# B&R Automation Studio project Parker_BMM_ST_V5_3147_V12 (part 12)

#### bdeflash.c
```c
/********************************************************************
 * COPYRIGHT --  B&R China
 ********************************************************************
 * Program: bdeflash
 * File: bdeflash.c
 * Author: lijianjun
 * Created: March 06, 2013
 ********************************************************************
 * Implementation of program bdeflash --- bottom deflasher control
 ********************************************************************/

#include <bur/plctypes.h>

#ifdef _DEFAULT_INCLUDES
	#include <AsDefault.h>
#endif

/**************************************************************************************
                            Function Declarations
**************************************************************************************/

//void BottomDeflash( Mold_typ * pMold);
void BottomDeflash( Mold_typ * pMold,TopDeflash_Fix_typ * pBottomDeflashFix, TopDeflash_Para_typ * pBottomDeflashPara,Mold_Para_User_typ * pMoldUser);
/**************************************************************************************
     	        		I N I T U P  O F   T H E   T A S K
**************************************************************************************/
_INIT void init ( void )
 {
 	LMold.BottomDeflash.Step = 0;
 	RMold.BottomDeflash.Step = 0;
 } /* end of _INIT */

 /*************************************************************************************
        		底部去飞边		C Y C L I C   P A R T   O F   T H E   T A S K
**************************************************************************************/

 _CYCLIC void cyclic ( void )
 {
 	if(!LMold.TimeSet.BottomDeflashBwAlarmTime)LMold.TimeSet.BottomDeflashBwAlarmTime = 1000;  /*  10s  */
 	if(!RMold.TimeSet.BottomDeflashBwAlarmTime)RMold.TimeSet.BottomDeflashBwAlarmTime = 1000;  /*  10s  */

 	LMold.TransDIn.BottomDeflashBwLimit = gMachineIn.LMold.BottomDeflashBwLimit;
 	LMold.TransDIn.BottomDeflashFwLimit = gMachineIn.LMold.BottomDeflashFwLimit;

	RMold.TransDIn.BottomDeflashBwLimit = gMachineIn.RMold.BottomDeflashBwLimit;
	RMold.TransDIn.BottomDeflashFwLimit = gMachineIn.RMold.BottomDeflashFwLimit;

	BottomDeflash(&LMold,&gMachineFix.MoldL.BottomDeflash,&gMachinePara.MoldL.BottomDeflash,&gUserPara.LMold);
	BottomDeflash(&RMold,&gMachineFix.MoldR.BottomDeflash,&gMachinePara.MoldR.BottomDeflash,&gUserPara.RMold);

//	gMachineOut.LMold.BottomDeflashFw = LMold.BottomDeflash.Out;
//	gMachineOut.RMold.BottomDeflashFw = RMold.BottomDeflash.Out;

	gMachineOut.LMold.BottomDeflashFw = LMold.ValveOut.BottomDeflashFw;
	gMachineOut.RMold.BottomDeflashFw = RMold.ValveOut.BottomDeflashFw;

	gMachineOut.LMold.BottomDeflashBw = LMold.ValveOut.BottomDeflashBw;
	gMachineOut.RMold.BottomDeflashBw = RMold.ValveOut.BottomDeflashBw;

	/*------------- ActuatorType--------------- */
	gMachineFix.MoldL.BottomDeflash.eActuatorType = gMachineFix.MoldR.BottomDeflash.eActuatorType;

	/*------------ PressueOutputType--------------- */
	gMachineFix.MoldL.BottomDeflash.ePressueOutputType = gMachineFix.MoldR.BottomDeflash.ePressueOutputType;

	/*------------ FluxOutputType--------------- */
	gMachineFix.MoldL.BottomDeflash.eFluxOutputType = gMachineFix.MoldR.BottomDeflash.eFluxOutputType;

 } /* end of _CYCLIC */

void BottomDeflash( Mold_typ * pMold,TopDeflash_Fix_typ * pBottomDeflashFix, TopDeflash_Para_typ * pBottomDeflashPara,Mold_Para_User_typ * pMoldUser)
{

	switch ( pMold->BottomDeflash.Step )
	{
		/*------------------ stop all the output ------------------*/
		case 0:
			pMold->BottomDeflash.Out      = 0;
			pMold->ActInfo.BottomDeflash  = 0;
			pMold->ActInfo.BottomDeflashFw  = 0;
			pMold->ActInfo.BottomDeflashBw  = 0;

			pMold->ValveOut.BottomDeflashFw = 0;

			if (0 == gMachineInfo.Auto)
			{
				pMold->ValveOut.BottomDeflashBw = 0;//ipis0726
			}

			pMold->BottomDeflash.Timer.IN	= 0;
			break;

		/*------------------ TopDeflash forward -------------------- */
		case 90: 			/* forward  Extra delay for Extrilift Acc charge */
			if(pMold->Option.BottomDeflash)
			{
				if(pMoldUser->TimeSet.BottomDeflashExtraDelay != 0)
				{
					pMold->BottomDeflash.Timer.IN = 1;
					pMold->BottomDeflash.Timer.PT = pMoldUser->TimeSet.BottomDeflashExtraDelay;
					pMold->BottomDeflash.Step 	= 95;
				}
				else
				{
					pMold->BottomDeflash.Step = 100;
				}
			}
			else
			{
				pMold->BottomDeflash.Step = 100;
			}

			break;

		case 95: 	/*Extara delay*/
			pMoldUser->TimeDis.BottomDeflashExtraDelay = pMold->BottomDeflash.Timer.ET;
			if (1 == pMold->BottomDeflash.Timer.Q)
			{
				pMold->BottomDeflash.Timer.IN       = 0;
				//	pMold->TimeDis.TopDeflashFwDelay = 0;
				pMold->BottomDeflash.Step = 100;
			}

			break;

		/*------------------ BottomDeflash forward -------------------- */
		case 100: /* BottomDeflash delay*/

			if(pMold->Option.BottomDeflash)
			{
				if(pMold->TimeSet.BottomDeflashFwDelay != 0)
				{
					pMold->BottomDeflash.Timer.IN = 1;
					pMold->BottomDeflash.Timer.PT = pMold->TimeSet.BottomDeflashFwDelay;
					pMold->BottomDeflash.Step 	= 200;
				}
				else
				{
					pMold->BottomDeflash.Step = 300;
				}
			}
			else
			{
				pMold->BottomDeflash.Step = 300;
			}
			break;

		case 200: 		/* delay ok */
			pMold->TimeDis.BottomDeflashFwDelay = pMold->BottomDeflash.Timer.ET;
			if (1 == pMold->BottomDeflash.Timer.Q)
			{
				pMold->BottomDeflash.Timer.IN       = 0;
				//	pMold->TimeDis.BottomDeflashFwDelay = 0;
				pMold->BottomDeflash.Step = 300;
			}
			break;

		case 300:
			if(pMold->Option.BottomDeflash)
			{
				switch (pBottomDeflashFix->eActuatorType )
				{
					/*-------------------------------------------------*/
					case ACTUATOR_HYD: /*1:Oil*/
					/*-------------------------------------------------*/
						if(pMold->TimeSet.BottomDeflashFwTime != 0 )
						{
							pMold->BottomDeflash.LimitTimer.IN = 1; //ipis0213
							pMold->BottomDeflash.LimitTimer.PT = pMold->TimeSet.BottomDeflashFwAlarmTime;

							pMold->BottomDeflash.Timer.IN = 1;
							pMold->BottomDeflash.Timer.PT = pMold->TimeSet.BottomDeflashFwTime;
							pMold->BottomDeflash.Step = 400;
						}
						else
						{
							//	pMold->BottomDeflash.Step = 499;
							pMold->BottomDeflash.Step = 2900; //ipis 0213
						}
						break;
					/*-------------------------------------------------*/
					case ACTUATOR_PNEU: /*2:Air*/
					/*-------------------------------------------------*/
						if(pMold->TimeSet.BottomDeflashFwTime != 0 )
						{
							pMold->BottomDeflash.Timer.IN = 1;
							pMold->BottomDeflash.Timer.PT = pMold->TimeSet.BottomDeflashFwTime;
							pMold->BottomDeflash.Step = 400;
						}
						else
						{
							//	pMold->BottomDeflash.Step = 499;
							pMold->BottomDeflash.Step = 2900; //ipis 0213
						}
						break;
				}
			}
			else
			{
				pMold->BottomDeflash.Step = 2900; // for no use
			}

			break;

		case 400:			/* forward time ok */
			pMold->BottomDeflash.Out     = 1;
			pMold->ActInfo.BottomDeflash = 1;
			pMold->ActInfo.BottomDeflashFw  = 1;
			pMold->ActInfo.BottomDeflashBw  = 0;

			pMold->ValveOut.BottomDeflashFw = 1;
			pMold->ValveOut.BottomDeflashBw = 0;

			pMold->BottomDeflash.p_set = pBottomDeflashPara->P_Fw;

			pMold->TimeDis.BottomDeflashFwTime = pMold->BottomDeflash.Timer.ET;

			if ((1 == pMold->BottomDeflash.Timer.Q) )
			{

				pMold->BottomDeflash.Out      = 0;
				pMold->ActInfo.BottomDeflashFw  = 0;
				pMold->ActInfo.BottomDeflashBw  = 0;

				pMold->ValveOut.BottomDeflashFw = 0;
				pMold->ValveOut.BottomDeflashBw = 0;

				pMold->BottomDeflash.p_set = 0;
				pMold->BottomDeflash.Timer.IN = 0;
				pMold->BottomDeflash.LimitTimer.IN = 0;
				//	pMold->TimeDis.BottomDeflashFwTime = 0;

				pMold->BottomDeflash.Step     = 410;

			}

			pMold->TimeDis.BottomDeflashFwAlarmTime = pMold->BottomDeflash.LimitTimer.ET;

			break;

		/*------------------------------------------------------------------------------*/

		case 410:/*Second Forward Delay*/

			switch (pBottomDeflashFix->eActuatorType)
			{
				/*-------------------------------------------------*/
				case ACTUATOR_HYD: /*1:Oil*/
				/*-------------------------------------------------*/
					if(pMoldUser->TimeSet.BottomDeflashSecDelay != 0)
					{
						pMold->BottomDeflash.Timer.IN = 1;
						pMold->BottomDeflash.Timer.PT = pMoldUser->TimeSet.BottomDeflashSecDelay;
						pMold->BottomDeflash.Step = 420;
					}
					else
					{
						pMold->BottomDeflash.Step = 430;
					}
					break;
				/*-------------------------------------------------*/
				case ACTUATOR_PNEU: /*2:Air*/
				/*-------------------------------------------------*/
					pMold->BottomDeflash.Step = 1300;
					break;
			}
			break;
		case 420: /*Start Second TopDeflash Forward Timer*/

			pMold->BottomDeflash.Out      = 0;
			pMold->ActInfo.BottomDeflashFw  = 0;
			pMold->ActInfo.BottomDeflashBw  = 0;

			pMold->ValveOut.BottomDeflashFw = 0;
			pMold->ValveOut.BottomDeflashBw = 0;

			pMold->BottomDeflash.p_set = 0;

			pMoldUser->TimeDis.BottomDeflashSecDelay = pMold->BottomDeflash.Timer.ET;
			if (1 == pMold->BottomDeflash.Timer.Q)
			{
				pMold->BottomDeflash.Timer.IN       = 0;
				pMold->BottomDeflash.LimitTimer.IN 	= 0;
				//	pMoldUser->TimeDis.BottomDeflashSecDelay = 0;
				pMold->BottomDeflash.Step = 430;
			}
			break;

		case 430:		/*Start Second TopDeflash Forward Timer*/
			if(pMoldUser->TimeSet.BottomDeflashSecTime != 0)
			{
				pMold->BottomDeflash.LimitTimer.IN = 1; //ipis0213
				pMold->BottomDeflash.LimitTimer.PT = pMold->TimeSet.BottomDeflashFwAlarmTime;

				pMold->BottomDeflash.Timer.IN = 1;
				pMold->BottomDeflash.Timer.PT = pMoldUser->TimeSet.BottomDeflashSecTime;
				pMold->BottomDeflash.Step = 440;
			}
			else
			{
				pMold->BottomDeflash.Step = 1300;
			}
			break;

		case 440:  /*Bottom deflash second forward */
			pMold->BottomDeflash.Out     = 1;
			pMold->ActInfo.BottomDeflash = 1;
			pMold->ActInfo.BottomDeflashFw  = 1;
			pMold->ActInfo.BottomDeflashBw  = 0;

			pMold->ValveOut.BottomDeflashFw = 1;
			pMold->ValveOut.BottomDeflashBw = 0;

			pMold->BottomDeflash.p_set = pBottomDeflashPara->P_Fw2nd;

			pMoldUser->TimeDis.BottomDeflashSecTime = pMold->BottomDeflash.Timer.ET;
			if ((1 == pMold->BottomDeflash.Timer.Q) || (1 == pMold->TransDIn.BottomDeflashFwLimit))
			{

				pMold->BottomDeflash.Out      = 0;
				pMold->ActInfo.BottomDeflashFw  = 0;
				pMold->ActInfo.BottomDeflashBw  = 0;

				pMold->ValveOut.BottomDeflashFw = 0;
				pMold->ValveOut.BottomDeflashBw = 0;
				pMold->BottomDeflash.p_set = 0;
				pMold->BottomDeflash.Timer.IN = 0;
				//	pMold->TimeDis.BottomDeflashFwTime = 0;
				//	pMoldUser->TimeDis.BottomDeflashSecTime=0;
				pMold->BottomDeflash.Step     = 1300;
			}
			pMold->TimeDis.BottomDeflashFwAlarmTime = pMold->BottomDeflash.LimitTimer.ET;

			break;

		/*----------------------------------------------*/
		/*No Time Movement-move unitl reach limit sensor*/
		/*----------------------------------------------*/

		case 499:
			pMold->BottomDeflash.Out     = 1;
			pMold->ActInfo.BottomDeflash = 1;
			pMold->ActInfo.BottomDeflashFw  = 1;
			pMold->ActInfo.BottomDeflashBw  = 0;

			pMold->ValveOut.BottomDeflashFw = 1;
			pMold->ValveOut.BottomDeflashBw = 0;

			pMold->BottomDeflash.p_set = pBottomDeflashPara->P_Fw;

			if (1 == pMold->TransDIn.BottomDeflashFwLimit)
			{

				pMold->BottomDeflash.Out      = 0;
				pMold->ActInfo.BottomDeflashFw  = 0;
				pMold->ActInfo.BottomDeflashBw  = 0;

				pMold->ValveOut.BottomDeflashFw = 0;
				pMold->ValveOut.BottomDeflashBw = 0;
				pMold->BottomDeflash.p_set = 0;
				pMold->BottomDeflash.Timer.IN = 0;
				pMold->BottomDeflash.LimitTimer.IN = 0;
				//	pMold->TimeDis.BottomDeflashFwTime = 0;

				pMold->BottomDeflash.Step     = 2900;
			}

			pMold->TimeDis.BottomDeflashFwAlarmTime = pMold->BottomDeflash.LimitTimer.ET;

			if (1 == pMold->BottomDeflash.LimitTimer.Q )
			{
				pMold->Alarm.BottomDeflashNotAtFwPos=1;
				pMold->BottomDeflash.Timer.IN   = 0;
				pMold->BottomDeflash.LimitTimer.IN = 0;
				pMold->BottomDeflash.Step = 40000;
			}

			break;

		case 1000:
			pMold->BottomDeflash.Out     = 1;
			pMold->ActInfo.BottomDeflashFw  = 1;
			pMold->ActInfo.BottomDeflashBw  = 0;
			pMold->BottomDeflash.p_set = pBottomDeflashPara->P_Fw;
			pMold->ValveOut.BottomDeflashFw = 1;
			pMold->ValveOut.BottomDeflashBw = 0;

			pMold->ActInfo.BottomDeflash = 1;
			break;

		/*------- BottomDeflash Bw --------------------------*/

		case 1300: /* BottomDeflash Bw delay*/
			if(pMold->Option.BottomDeflash)
			{
				switch (pBottomDeflashFix->eActuatorType)
				{
					/*-------------------------------------------------*/
					case ACTUATOR_HYD: /*1:Oil*/
					/*-------------------------------------------------*/
						if(pMold->TimeSet.BottomDeflashBwDelay != 0)
						{
							pMold->BottomDeflash.Timer.IN = 1;
							pMold->BottomDeflash.Timer.PT = pMold->TimeSet.BottomDeflashBwDelay;
							pMold->BottomDeflash.Step 	= 1400;
						}
						else
						{
							pMold->BottomDeflash.Step = 1500;
						}

						break;
					/*-------------------------------------------------*/
					case ACTUATOR_PNEU: /*2:Air*/
					/*-------------------------------------------------*/
						pMold->BottomDeflash.Step = 1500;
						break;
				}
			}
			else
			{
				pMold->BottomDeflash.Step = 1500;
			}
			break;
		case 1400: /* delay ok */
			pMold->TimeDis.BottomDeflashBwDelay = pMold->BottomDeflash.Timer.ET;
			if (1 == pMold->BottomDeflash.Timer.Q)
			{
				pMold->BottomDeflash.Timer.IN       = 0;
				//		pMold->TimeDis.BottomDeflashBwDelay = 0;
				pMold->BottomDeflash.Step = 1500;
			}
			break;

		case 1500:

			if(pMold->Option.BottomDeflash)
			{
				pMold->BottomDeflash.Timer.IN = 1;
				pMold->BottomDeflash.Timer.PT = pMold->TimeSet.BottomDeflashBwAlarmTime;
				pMold->BottomDeflash.Step = 1600;
			}
			else
			{
				pMold->BottomDeflash.Step = 1700; // for no use
			}
			break;

		case 1600:
			pMold->BottomDeflash.Out     = 0;

			pMold->ActInfo.BottomDeflash = 0;
			pMold->ActInfo.BottomDeflashFw  = 0;
			pMold->ActInfo.BottomDeflashBw  = 1;

			pMold->ValveOut.BottomDeflashFw = 0;
			pMold->ValveOut.BottomDeflashBw = 1;

			pMold->BottomDeflash.p_set = pBottomDeflashPara->P_Bw;

			pMold->TimeDis.BottomDeflashBwAlarmTime = pMold->BottomDeflash.Timer.ET;

			if (1 == pMold->TransDIn.BottomDeflashBwLimit)
			{
				pMold->BottomDeflash.Out      = 0;
				pMold->ActInfo.BottomDeflashFw  = 0;
				pMold->ActInfo.BottomDeflashBw  = 0;

				pMold->ValveOut.BottomDeflashFw = 0;
				pMold->ValveOut.BottomDeflashBw = 0;
				pMold->BottomDeflash.p_set=0;

				pMold->BottomDeflash.Timer.IN = 0;
				pMold->TimeDis.BottomDeflashBwTime = 0;
				pMold->BottomDeflash.Step     = 2900;
			}

			break;

		case 1700: // for no use

			if (1 == pMold->TransDIn.BottomDeflashBwLimit)
			{
				pMold->BottomDeflash.Out      = 0;
				pMold->ActInfo.BottomDeflashFw  = 0;
				pMold->ActInfo.BottomDeflashBw  = 0;

				pMold->ValveOut.BottomDeflashFw = 0;
				pMold->ValveOut.BottomDeflashBw = 0;
				pMold->BottomDeflash.p_set=0;

				pMold->BottomDeflash.Timer.IN = 0;
				pMold->TimeDis.BottomDeflashBwTime = 0;
				pMold->BottomDeflash.Step     = 2900;
			}
			else
			{
				pMold->BottomDeflash.Timer.IN   = 0;
				pMold->Alarm.BottomDeflashNotAtBwPos = 1;
				pMold->BottomDeflash.Step = 40000;           /*  TopDeflash backward alarm   */

			}

			//			pMold->TimeDis.BottomDeflashBwAlarmTime = pMold->BottomDeflash.Timer.ET;
			//			if(1 == pMold->BottomDeflash.Timer.Q)
			//			{
			//				pMold->ValveOut.BottomDeflashFw  = 0;
			//				pMold->ValveOut.BottomDeflashBw  = 0;
			//
			//				pMold->BottomDeflash.Timer.IN   = 0;
			//				pMold->Alarm.BottomDeflashNotAtBwPos = 1;
			//				pMold->BottomDeflash.Step = 40000;           /*  TopDeflash backward alarm   */
			//			}

			break;
		/*----------for handle bottom deflash force backward------------------------------*/
		case 1950: //for auto force backward

			pMold->BottomDeflash.Timer.IN = 0;
			pMold->BottomDeflash.LimitTimer.IN = 0;
			pMold->BottomDeflash.Step = 2000;

			break;

		case 2000:
			pMold->BottomDeflash.Out     = 0;
			pMold->ActInfo.BottomDeflash = 0;
			pMold->ActInfo.BottomDeflashFw  = 0;
			pMold->ActInfo.BottomDeflashBw  = 0;
			pMold->BottomDeflash.p_set=0;
			pMold->ValveOut.BottomDeflashFw = 0;
			pMold->ValveOut.BottomDeflashBw = 0;

			pMold->BottomDeflash.Step    = 0;
			break;

		case 2900:

			pMold->BottomDeflash.Timer.IN = 0;
			pMold->BottomDeflash.LimitTimer.IN = 0;
			pMold->BottomDeflash.Out     = 0;
			pMold->ActInfo.BottomDeflashFw  = 0;
			pMold->ActInfo.BottomDeflashBw  = 0;
			pMold->BottomDeflash.p_set=0;

			pMold->ValveOut.BottomDeflashFw = 0;
			pMold->ValveOut.BottomDeflashBw = 0;
			pMold->ActInfo.BottomDeflash = 0;
			pMold->BottomDeflash.Step    = 3000;
			break;

		case 3000:
			break;

		case 5000: /* FW*/

			//			pMold->ActInfo.BottomDeflashFw  = 1;
			//			pMold->ActInfo.BottomDeflashBw  = 0;
			//
			//			pMold->ValveOut.BottomDeflashFw = 1;
			//			pMold->ValveOut.BottomDeflashBw = 0;
			//
			//			pMold->BottomDeflash.p_set = pBottomDeflashPara->P_CalibFw;

			if(0 == pMold->TransDIn.BottomDeflashFwLimit)
			{
				pMold->ActInfo.BottomDeflashFw  = 1;
				pMold->ActInfo.BottomDeflashBw  = 0;

				pMold->ValveOut.BottomDeflashFw = 1;
				pMold->ValveOut.BottomDeflashBw = 0;

				pMold->BottomDeflash.p_set = pBottomDeflashFix->pCalibMax;
				pMold->BottomDeflash.v_set = pBottomDeflashFix->vCalibMax;
			}
			else
			{
				pMold->ActInfo.BottomDeflashFw  = 0;
				pMold->ActInfo.BottomDeflashBw  = 0;

				pMold->ValveOut.BottomDeflashFw = 0;
				pMold->ValveOut.BottomDeflashBw = 0;

				pMold->BottomDeflash.p_set 		= 0;
				pMold->BottomDeflash.v_set		= 0;

				pMold->BottomDeflash.Step    	= 20000;
			}

			break;

		case 15000: /* BW*/

			//			pMold->ActInfo.BottomDeflashFw  = 0;
			//			pMold->ActInfo.BottomDeflashBw  = 1;
			//
			//			pMold->ValveOut.BottomDeflashFw = 0;
			//			pMold->ValveOut.BottomDeflashBw = 1;
			//
			//			pMold->BottomDeflash.p_set = pBottomDeflashPara->P_CalibBw;

			if(0 == pMold->TransDIn.BottomDeflashBwLimit)
			{
				pMold->ActInfo.BottomDeflashFw  = 0;
				pMold->ActInfo.BottomDeflashBw  = 1;

				pMold->ValveOut.BottomDeflashFw = 0;
				pMold->ValveOut.BottomDeflashBw = 1;

				pMold->BottomDeflash.p_set = pBottomDeflashFix->pCalibZero;
				pMold->BottomDeflash.v_set = pBottomDeflashFix->vCalibZero;

			}
			else

			{
				pMold->ActInfo.BottomDeflashFw  = 0;
				pMold->ActInfo.BottomDeflashBw  = 0;

				pMold->ValveOut.BottomDeflashFw = 0;
				pMold->ValveOut.BottomDeflashBw = 0;

				pMold->BottomDeflash.p_set 		= 0;
				pMold->BottomDeflash.v_set 		= 0;
				pMold->BottomDeflash.Step    = 20000;
			}

			break;

		/*--------------- Manual action stop -----------------*/
		case 20000:

			pMold->BottomDeflash.Out      = 0;

			pMold->BottomDeflash.Timer.IN   = 0;
			pMold->BottomDeflash.LimitTimer.IN = 0;
			pMold->ActInfo.BottomDeflashFw  = 0;
			pMold->ActInfo.BottomDeflashBw  = 0;

			pMold->ValveOut.BottomDeflashFw = 0;
			pMold->ValveOut.BottomDeflashBw = 0;

			pMold->BottomDeflash.p_set		= 0;
			pMold->BottomDeflash.v_set 		= 0;

			pMold->BottomDeflash.Step 	 	= 0;
			break;

		/*--------------- Instance stop -----------------*/
		case 30000:
			pMold->BottomDeflash.Out      = 0;

			pMold->BottomDeflash.Timer.IN   = 0;
			pMold->BottomDeflash.LimitTimer.IN = 0;

			pMold->ActInfo.BottomDeflashFw  = 0;
			pMold->ActInfo.BottomDeflashBw  = 0;

			pMold->ValveOut.BottomDeflashFw = 0;
			pMold->ValveOut.BottomDeflashBw = 0;

			pMold->BottomDeflash.p_set		= 0;
			pMold->BottomDeflash.v_set 		= 0;

			pMold->BottomDeflash.Step     	= 0;
			break;

		/*--------------- error -----------------*/
		case 40000:
			pMold->BottomDeflash.Out      = 0;

			pMold->BottomDeflash.Timer.IN   = 0;
			pMold->BottomDeflash.LimitTimer.IN = 0;

			pMold->ActInfo.BottomDeflashFw  = 0;
			pMold->ActInfo.BottomDeflashBw  = 0;

			pMold->ValveOut.BottomDeflashFw = 0;
			pMold->ValveOut.BottomDeflashBw = 0;
			pMold->BottomDeflash.p_set		= 0;
			pMold->BottomDeflash.v_set 		= 0;
			break;
	}/* end of switch */

	/* ----------------- BottomDeflash Fw / Bw timeout --------------------  */
	if(1 == pMold->BottomDeflash.LimitTimer.Q && 1 == gMachineInfo.TimeLimit)
	{
		if(pMold->BottomDeflash.Step < 500 && pMold->BottomDeflash.Step > 300)		/* BottomDeflash Fw  */
		{
			pMold->Alarm.BottomDeflashNotAtFwPos = 1;
		}

		if(pMold->BottomDeflash.Step < 1700 && pMold->BottomDeflash.Step > 1400)	/* BottomDeflash Bw  */
		{
			pMold->Alarm.BottomDeflashNotAtBwPos = 1;
		}

		pMold->BottomDeflash.Timer.IN   = 0;
		pMold->BottomDeflash.LimitTimer.IN = 0;
		pMold->BottomDeflash.Step = 40000;

	}

	/* ----------------- BottomDeflash action limit --------------------  */
	if(pMold->BottomDeflash.Step > 100 && pMold->BottomDeflash.Step < 500)
	{
		if(0 == pMold->Clamp.ClsPos)
		{
			pMold->Alarm.ClampNotAtClsDI  = !pMold->Clamp.ClsPos;
			pMold->TopDeflash.Step = 40000;
		}

		if(0 == pMold->Carriage.BwPos)
		{
			pMold->Alarm.CarriageNotAtBwDI = !pMold->Carriage.BwPos;
			pMold->TopDeflash.Step = 40000;
		}
	}

	if((pMold->BottomDeflash.Step > 1300 && pMold->BottomDeflash.Step < 1700))
	{

	}

}/*end of function */
```

### Program Logical/process/tdeflash (ANSIC, version 1.00.0) - top deflash

#### tdeflash.c
```c
/********************************************************************
 * COPYRIGHT --  B&R China
 ********************************************************************
 * Program: tdeflash
 * File: tdeflash.c
 * Author: lijianjun
 * Created: March 06, 2013
 ********************************************************************
 * Implementation of program tdeflash --- top deflasher control
 ********************************************************************/

#include <bur/plctypes.h>

#ifdef _DEFAULT_INCLUDES
#include <AsDefault.h>
#endif

/**************************************************************************************
                            Function Declarations
**************************************************************************************/

//void TopDeflash( Mold_typ * pMold, Punch_Para_typ * pTopDeflashPara);
void TopDeflash( Mold_typ * pMold, TopDeflash_Fix_typ * pTopDeflashFix, TopDeflash_Para_typ * pTopDeflashPara,Mold_Para_User_typ * pMoldUser);

/**************************************************************************************
     	        		I N I T U P  O F   T H E   T A S K
**************************************************************************************/
_INIT void init ( void )
{
	LMold.TopDeflash.Step = 30000;
	RMold.TopDeflash.Step = 30000;
} /* end of _INIT */

 /*************************************************************************************
        				C Y C L I C   P A R T   O F   T H E   T A S K
**************************************************************************************/

_CYCLIC void cyclic ( void )
{
	if(!LMold.TimeSet.TopDeflashFwAlarmTime)LMold.TimeSet.TopDeflashFwAlarmTime = 1000;  /*  10s  */
	if(!RMold.TimeSet.TopDeflashFwAlarmTime)RMold.TimeSet.TopDeflashFwAlarmTime = 1000;  /*  10s  */

	if(!LMold.TimeSet.TopDeflashBwAlarmTime)LMold.TimeSet.TopDeflashBwAlarmTime = 1000;  /*  10s  */
	if(!RMold.TimeSet.TopDeflashBwAlarmTime)RMold.TimeSet.TopDeflashBwAlarmTime = 1000;  /*  10s  */

	if(!LMold.TimeSet.TopDeflashOpnAlarmTime)LMold.TimeSet.TopDeflashOpnAlarmTime = 1000;  /*  10s  */
	if(!RMold.TimeSet.TopDeflashOpnAlarmTime)RMold.TimeSet.TopDeflashOpnAlarmTime = 1000;  /*  10s  */

	LMold.TransDIn.TopDeflashBwLimit = gMachineIn.LMold.TopDeflashBwLimit;
	LMold.TransDIn.TopDeflashFwLimit = gMachineIn.LMold.TopDeflashFwLimit;

	RMold.TransDIn.TopDeflashBwLimit = gMachineIn.RMold.TopDeflashBwLimit;
	RMold.TransDIn.TopDeflashFwLimit = gMachineIn.RMold.TopDeflashFwLimit;

	LMold.TransDIn.TopDeflashOpnLimit = gMachineIn.LMold.TopDeflashOpnLimit;
	RMold.TransDIn.TopDeflashOpnLimit = gMachineIn.RMold.TopDeflashOpnLimit;

	TopDeflash(&LMold,&gMachineFix.MoldL.TopDeflash,&gMachinePara.MoldL.TopDeflash,&gUserPara.LMold);
	TopDeflash(&RMold,&gMachineFix.MoldR.TopDeflash,&gMachinePara.MoldR.TopDeflash,&gUserPara.RMold);

	gMachineOut.LMold.TopDeflashFw  = LMold.ValveOut.TopDeflashFw;
	gMachineOut.LMold.TopDeflashBw  = LMold.ValveOut.TopDeflashBw;

	gMachineOut.LMold.TopDeflashCls = LMold.ValveOut.TopDeflashCls;

	gMachineOut.RMold.TopDeflashFw  = RMold.ValveOut.TopDeflashFw;
	gMachineOut.RMold.TopDeflashBw  = RMold.ValveOut.TopDeflashBw;

	gMachineOut.RMold.TopDeflashCls = RMold.ValveOut.TopDeflashCls;

	gMachineOut.RMold.TopDeflashCool = RMold.ValveOut.TopDeflashCool;
	gMachineOut.LMold.TopDeflashCool = LMold.ValveOut.TopDeflashCool;

	/*------------- ActuatorType--------------- */
	gMachineFix.MoldL.TopDeflash.eActuatorType = gMachineFix.MoldR.TopDeflash.eActuatorType;

	/*------------ PressueOutputType--------------- */
	gMachineFix.MoldL.TopDeflash.ePressueOutputType = gMachineFix.MoldR.TopDeflash.ePressueOutputType;

	/*------------ FluxOutputType--------------- */
	gMachineFix.MoldL.TopDeflash.eFluxOutputType = gMachineFix.MoldR.TopDeflash.eFluxOutputType;

} /* end of _CYCLIC */

void TopDeflash( Mold_typ * pMold,TopDeflash_Fix_typ * pTopDeflashFix, TopDeflash_Para_typ * pTopDeflashPara,Mold_Para_User_typ * pMoldUser)
{

	switch ( pMold->TopDeflash.Step )
	{
		/*------------------ stop all the output ------------------*/
		case 0:

			pMold->ValveOut.TopDeflashCool = 0;/*Albert*/

			//			if(1 == gMachineInfo.Auto)
			//			{
			//				pMold->ValveOut.TopDeflashFw = 0;
			//				pMold->ValveOut.TopDeflashBw = 1;
			//			}

			pMold->ActInfo.TopDeflashPuncher = 0;
			//	pMold->ActInfo.TopDeflashFw = pMold->ValveOut.TopDeflashFw;
			//	pMold->ActInfo.TopDeflashBw = pMold->ValveOut.TopDeflashBw;
			pMold->ActInfo.TopDeflashFw = 0;
			pMold->ActInfo.TopDeflashBw = 0;

			if (0 == gMachineInfo.Auto) //ipis0726
			{
				pMold->ValveOut.TopDeflashBw = 0;
			}

			pMold->TopDeflash.p_set = 0;
			pMold->TopDeflash.v_set = 0;

			pMold->TopDeflash.Timer.IN	= 0;
			break;

		/*------------------ TopDeflash prepare forward -------------------- */
		case 10:			/* TopDeflash prepare forward */
			if(pMold->Option.TopDeflash)
			{
				pMold->TopDeflash.Timer.IN = 1;
				pMold->TopDeflash.Timer.PT = pMold->TimeSet.TopDeflashPreFwTime;
				pMold->TopDeflash.Step = 20;
			}
			else
			{
				pMold->TopDeflash.Step = 30;
			}
			break;

		case 20:

			pMold->ActInfo.TopDeflashFw = 1;
			pMold->ActInfo.TopDeflashBw = 0;

			pMold->ValveOut.TopDeflashFw  = 1;
			pMold->ValveOut.TopDeflashBw  = 0;
			pMold->ValveOut.TopDeflashCls = 0;

			pMold->TopDeflash.p_set = pTopDeflashPara->P_Fw;/*Albert*/

			pMold->TimeDis.TopDeflashPreFwTime = pMold->TopDeflash.Timer.ET;
			if (1 == pMold->TopDeflash.Timer.Q )
			{
				pMold->ValveOut.TopDeflashFw  = 0;
				pMold->ValveOut.TopDeflashBw  = 0;
				pMold->ValveOut.TopDeflashCls = 0;

				pMold->TopDeflash.Timer.IN = 0;
				pMold->TimeDis.TopDeflashPreFwTime = 0;

				//		pMold->CoolDeflash.Step = 100;		/* cooling deflash  */ //ipis0731
				pMold->TopDeflash.Step = 30;
			}

			if (1 == pMold->TransDIn.TopDeflashFwLimit)
			{
				pMold->ValveOut.TopDeflashFw = 0;
				pMold->TopDeflash.Timer.IN   = 0;
				pMold->TimeDis.TopDeflashPreFwTime = 0;
				pMold->TopDeflash.Step = 40000;
			}
			break;

		case 30:
			if(0 == pMold->Option.CoolPin)
			{
				pMold->TopDeflash.Step = 100;	/*  defalsh forward */
			}

			if(0 == pMold->Option.TopDeflash)
			{
				pMold->CoolPin.Step     = 100;	/*  cool pin down    */
				pMold->CoolPinBlow.Step = 100;	/*  cool pin blowing  */
			}

			if(1 == pMold->Option.CoolPin && 1 == pMold->Option.TopDeflash)
			{
				if( 0 == pMold->Option.PunchHandle)
				{
					pMold->CoolPin.Step     = 100;/*  cool pin down      */
					pMold->CoolPinBlow.Step = 100;/*  cool pin blowing  */
				}
				else
				{
					pMold->TopDeflash.Step = 100;/*  defalsh forward    */
				}
			}
			break;

		/*------------------ TopDeflash forward -------------------- */
		case 90: 			/* forward  Extra delay for Extrilift Acc charge */
			if(pMold->Option.TopDeflash)
			{
				if(pMoldUser->TimeSet.TopDeflashExtraDelay != 0)
				{
					pMold->TopDeflash.Timer.IN = 1;
					pMold->TopDeflash.Timer.PT = pMoldUser->TimeSet.TopDeflashExtraDelay;
					pMold->TopDeflash.Step 	= 95;
				}
				else
				{
					pMold->TopDeflash.Step = 100;
				}
			}
			else
			{
				pMold->TopDeflash.Step = 100;
			}

			break;

		case 95: 	/*Extara delay*/
			pMoldUser->TimeDis.TopDeflashExtraDelay = pMold->TopDeflash.Timer.ET;
			if (1 == pMold->TopDeflash.Timer.Q)
			{
				pMold->TopDeflash.Timer.IN       = 0;
				//	pMold->TimeDis.TopDeflashFwDelay = 0;
				pMold->TopDeflash.Step = 100;
			}

			break;

		/*-------------------------------------- */
		case 100: 			/* forward delay*/
			//		pMold->ValveOut.TopDeflashFw  = 0;
			//		pMold->ValveOut.TopDeflashBw  = 0;
			//		pMold->ValveOut.TopDeflashCls = 0;
			//

			pMold->CutNeck.Step = 100;   	/* 旋切瓶口 */
			pMold->CoolDeflash.Step =100; 	/* 打手把吹冷*/
			if(pMold->Option.TopDeflash)
			{
				//		pMold->CoolDeflash.Step = 100;		/* cooling deflash  */ //ipis0731
				if(pMold->TimeSet.TopDeflashFwDelay != 0)
				{
					pMold->TopDeflash.Timer.IN = 1;
					pMold->TopDeflash.Timer.PT = pMold->TimeSet.TopDeflashFwDelay;
					pMold->TopDeflash.Step 	= 200;

					//gExSPC
					if(pMold == & LMold)
					{
						gExSPC[ExIndex].LMold.TopDeflashFwDelay = pMold->TimeSet.TopDeflashFwDelay/100.0;
					}
					else
					{
						gExSPC[ExIndex].RMold.TopDeflashFwDelay = pMold->TimeSet.TopDeflashFwDelay/100.0;
					}
				}
				else
				{
					pMold->TopDeflash.Step = 300;
				}
			}
			else
			{
				//	pMold->ActInfo.TopDeflashFw = 0;
				//	pMold->ActInfo.TopDeflashBw = 0;
				pMold->TopDeflash.Step = 300;
			}
			break;

		case 200: 			/* forward delay ok */
			pMold->TimeDis.TopDeflashFwDelay = pMold->TopDeflash.Timer.ET;
			if (1 == pMold->TopDeflash.Timer.Q)
			{
				pMold->TopDeflash.Timer.IN       = 0;
				//	pMold->TimeDis.TopDeflashFwDelay = 0;
				pMold->TopDeflash.Step = 300;
			}
			break;

		case 300:

			if(pMold->Option.TopDeflash)
			{
				switch (pTopDeflashFix->eActuatorType)
				{
					/*-------------------------------------------------*/
					case ACTUATOR_HYD: /*1:Oil*/
						/*-------------------------------------------------*/
						if(pMold->TimeSet.TopDeflashFwTime != 0)
						{
							pMold->TopDeflash.LimitTimer.IN = 1; //ipis0213
							pMold->TopDeflash.LimitTimer.PT = pMold->TimeSet.TopDeflashFwAlarmTime;

							pMold->TopDeflash.Timer.IN = 1;
							pMold->TopDeflash.Timer.PT = pMold->TimeSet.TopDeflashFwTime;
							pMold->TopDeflash.Step = 400;

							//gExSPC
							if(pMold == & LMold)
							{
								gExSPC[ExIndex].LMold.TopDeflashFwTime = pMold->TimeSet.TopDeflashFwTime/100.0;
							}
							else
							{
								gExSPC[ExIndex].RMold.TopDeflashFwTime = pMold->TimeSet.TopDeflashFwTime/100.0;
							}
						}
						else
						{
							//	pMold->TopDeflash.Step = 499;/*If no timer then direct forward until reach limit sensor*/
							//							pMold->TopDeflash.Step = 2900;/*If no timer then direct forward until reach limit sensor*/ //ipis2190131
							pMold->TopDeflash.Step = 410;
						}
						break;
					/*-------------------------------------------------*/
					case ACTUATOR_PNEU: /*2:Air*/
						/*-------------------------------------------------*/
						if(pMold->TimeSet.TopDeflashFwTime != 0 )
						{
							pMold->TopDeflash.Timer.IN = 1;
							pMold->TopDeflash.Timer.PT = pMold->TimeSet.TopDeflashFwTime;
							pMold->TopDeflash.Step = 400;
						}
						else
						{
							//	pMold->TopDeflash.Step = 499;
							pMold->TopDeflash.Step = 2900; //ipis 0213
						}
						break;
				}
			}
			else
			{
				pMold->TopDeflash.Step = 2900;  // for no use
			}
			break;

		case 400:			/* forward time ok */
			pMold->ActInfo.TopDeflashFw = 1;
			pMold->ActInfo.TopDeflashBw = 0;

			pMold->ValveOut.TopDeflashFw  = 1;
			pMold->ValveOut.TopDeflashBw  = 0;
			pMold->ValveOut.TopDeflashCls = 0;

			pMold->TopDeflash.p_set = pTopDeflashPara->P_Fw;/*Albert*/
			pMold->TopDeflash.v_set = pTopDeflashPara->V_Fw;

			pMold->TimeDis.TopDeflashFwTime = pMold->TopDeflash.Timer.ET;

			if (1 == pMold->TopDeflash.Timer.Q || (1 == pMold->TransDIn.TopDeflashFwLimit))
			{

				//gExSPC
				if(pMold == & LMold)
				{
					gExSPC[ExIndex].LMold.tTopDeflash1 = pMold->TopDeflash.LimitTimer.ET/100.0;
				}
				else
				{
					gExSPC[ExIndex].RMold.tTopDeflash1 = pMold->TopDeflash.LimitTimer.ET/100.0;
				}

				pMold->ValveOut.TopDeflashFw = 0;
				pMold->TopDeflash.Timer.IN   = 0;
				pMold->TopDeflash.LimitTimer.IN = 0;
				//			pMold->TimeDis.TopDeflashFwTime = 0;

				pMold->TopDeflash.p_set = 0;/*Albert*/
				pMold->TopDeflash.v_set = 0;

				pMold->TopDeflash.Step = 410;

			}

			pMold->TimeDis.TopDeflashFwAlarmTime = pMold->TopDeflash.LimitTimer.ET;

			//			if (1 == pMold->TopDeflash.LimitTimer.Q )
			//			{
			//
			//				pMold->Alarm.TopDeflashNotAtFwPos=1;
			//				pMold->TopDeflash.Timer.IN   = 0;
			//				pMold->TopDeflash.LimitTimer.IN = 0;
			//				pMold->TopDeflash.Step = 40000;
			//			}

			break;

		case 410:/*Second Forward Delay*/

			switch (pTopDeflashFix->eActuatorType)
			{
				/*-------------------------------------------------*/
				case ACTUATOR_HYD: /*1:Oil*/
					/*-------------------------------------------------*/
					if(pMoldUser->TimeSet.TopDeflashSecDelay != 0)
					{
						pMold->TopDeflash.Timer.IN = 1;
						pMold->TopDeflash.Timer.PT = pMoldUser->TimeSet.TopDeflashSecDelay;
						pMold->TopDeflash.Step = 420;

						//gExSPC
						if(pMold == & LMold)
						{
							gExSPC[ExIndex].LMold.TopDeflashSecDelay = pMoldUser->TimeSet.TopDeflashSecDelay/100.0;
						}
						else
						{
							gExSPC[ExIndex].RMold.TopDeflashSecDelay = pMoldUser->TimeSet.TopDeflashSecDelay/100.0;
						}
					}
					else
					{
						pMold->CoolDeflash.Step = 450;  //ipis0731
						pMold->TopDeflash.Step = 430;
					}

					break;
				/*-------------------------------------------------*/
				case ACTUATOR_PNEU: /*2:Air*/
					/*-------------------------------------------------*/
					pMold->CoolDeflash.Step = 450;  //ipis0731
					if(1 == gMachineInfo.Auto)
					{
						pMold->TopDeflash.Step = 500;
					}
					else
					{
						pMold->TopDeflash.Step = 2900;
					}

					break;
			}

			break;
		case 420:/*wait delay for cool deflash*/
			pMold->ActInfo.TopDeflashFw = 0;
			pMold->ActInfo.TopDeflashBw = 0;

			pMold->ValveOut.TopDeflashFw  = 0;
			pMold->ValveOut.TopDeflashBw  = 0;
			pMold->ValveOut.TopDeflashCls = 0;

			pMold->TopDeflash.p_set = 0;/*Albert*/
			pMold->ValveOut.TopDeflashCool = 1;

			pMoldUser->TimeDis.TopDeflashSecDelay = pMold->TopDeflash.Timer.ET;
			if(pMold->TopDeflash.Timer.Q)
			{
				pMold->TopDeflash.Timer.IN = 0;
				pMold->TopDeflash.LimitTimer.IN = 0;
				//	pMoldUser->TimeDis.TopDeflashSecDelay =0;
				pMold->TopDeflash.Step = 430;
			}
			break;

		case 430:/*Start Second TopDeflash Forward Timer*/

			if(pMoldUser->TimeSet.TopDeflashSecTime != 0)
			{
				pMold->TopDeflash.LimitTimer.IN = 1;  //ipis0213
				pMold->TopDeflash.LimitTimer.PT = pMold->TimeSet.TopDeflashFwAlarmTime;

				pMold->TopDeflash.Timer.IN = 1;
				pMold->TopDeflash.Timer.PT = pMoldUser->TimeSet.TopDeflashSecTime;
				pMold->TopDeflash.Step = 440;

				//gExSPC
				if(pMold == & LMold)
				{
					gExSPC[ExIndex].LMold.TopDeflashSecTime = pMoldUser->TimeSet.TopDeflashSecTime/100.0;
				}
				else
				{
					gExSPC[ExIndex].RMold.TopDeflashSecTime = pMoldUser->TimeSet.TopDeflashSecTime/100.0;
				}
			}
			else
			{
				pMold->TopDeflash.Step = 500;
			}

			break;
		case 440:/*Topdeflash second forward */
			pMold->ActInfo.TopDeflashFw = 1;
			pMold->ActInfo.TopDeflashBw = 0;

			pMold->ValveOut.TopDeflashFw  = 1;
			pMold->ValveOut.TopDeflashBw  = 0;
			pMold->ValveOut.TopDeflashCls = 0;

			pMold->ValveOut.TopDeflashCool = 1;/*Albert*/

			pMold->TopDeflash.p_set = pTopDeflashPara->P_Fw2nd;/*Albert*/
			pMold->TopDeflash.v_set = pTopDeflashPara->V_Fw2nd;/*Albert*/

			pMoldUser->TimeDis.TopDeflashSecTime = pMold->TopDeflash.Timer.ET;

			if (1== pMold->Option.PunchHandle)
			{
				if ((1 == pMold->TopDeflash.Timer.Q )|| (1 == pMold->TransDIn.TopDeflashFwLimit))
				{
					pMold->ValveOut.TopDeflashFw = 0;
					pMold->ValveOut.TopDeflashCool = 0;/*Albert*/
					//					pMold->CoolDeflash.Step =500; //ipis0731  //owen1021
					pMold->TopDeflash.Timer.IN   = 0;
					pMold->TopDeflash.LimitTimer.IN = 0;
					//	pMoldUser->TimeDis.TopDeflashSecTime =0;
					pMold->TopDeflash.p_set = 0;/*Albert*/
					pMold->TopDeflash.v_set = 0;
					pMold->TopDeflash.Step = 450;
					//				if ((1 == pMold->TransDIn.TopDeflashFwLimit))
					//				{
					//					if(1 == gMachineInfo.Auto)
					//					{
					//						pMold->TopDeflash.Step = 500;
					//					}
					//					else
					//					{
					//						pMold->TopDeflash.Step = 2900;
					//					}
					//				}

				}
			}
			else
			{
				if ((1 == pMold->TopDeflash.Timer.Q )||(1 == pMold->TransDIn.TopDeflashFwLimit))
				{
					//gExSPC
					if(pMold == & LMold)
					{
						gExSPC[ExIndex].LMold.tTopDeflash2 = pMold->TopDeflash.LimitTimer.ET/100.0;
					}
					else
					{
						gExSPC[ExIndex].RMold.tTopDeflash2 = pMold->TopDeflash.LimitTimer.ET/100.0;
					}

					pMold->ValveOut.TopDeflashFw = 0;
					pMold->ValveOut.TopDeflashCool = 0;/*Albert*/
					pMold->TopDeflash.Timer.IN   = 0;
					pMold->TopDeflash.LimitTimer.IN = 0;
					//	pMoldUser->TimeDis.TopDeflashSecTime =0;
					pMold->TopDeflash.p_set = 0;/*Albert*/
					pMold->TopDeflash.Step = 450;

					if(1 == gMachineInfo.Auto)
					{
						pMold->TopDeflash.Step = 500;
					}
					else
					{
						pMold->TopDeflash.Step = 2900;
					}

				}

			}

			pMold->TimeDis.TopDeflashFwAlarmTime = pMold->TopDeflash.LimitTimer.ET;

			//			if (1 == pMold->TopDeflash.LimitTimer.Q )
			//			{
			//				pMold->ValveOut.TopDeflashFw = 0;
			//				pMold->ValveOut.TopDeflashCool = 0;/*Albert*/
			//				pMold->CoolDeflash.Step =500; //ipis0731
			//				pMold->TopDeflash.p_set = 0;/*Albert*/
			//
			//				pMold->Alarm.TopDeflashNotAtFwPos=1;
			//				pMold->TopDeflash.Timer.IN   = 0;
			//				pMold->TopDeflash.LimitTimer.IN = 0;
			//				pMold->TopDeflash.Step = 40000;
			//			}

			break;

		case 450:

			if ((1 == pMold->TransDIn.TopDeflashFwLimit))
			{
				if(1 == gMachineInfo.Auto)
				{
					pMold->TopDeflash.Step = 500;
				}
				else
				{
					pMold->TopDeflash.Step = 2900;
				}
			}
			pMold->TimeDis.TopDeflashFwAlarmTime = pMold->TopDeflash.LimitTimer.ET;

			//			if (1 == pMold->TopDeflash.LimitTimer.Q )
			//			{
			//				pMold->ValveOut.TopDeflashFw = 0;
			//				pMold->ValveOut.TopDeflashCool = 0;/*Albert*/
			//				pMold->CoolDeflash.Step =500; //ipis0731
			//				pMold->TopDeflash.p_set = 0;/*Albert*/
			//
			//				pMold->Alarm.TopDeflashNotAtFwPos=1;
			//				pMold->TopDeflash.Timer.IN   = 0;
			//				pMold->TopDeflash.LimitTimer.IN = 0;
			//				pMold->TopDeflash.Step = 40000;
			//			}

			break;

		/*----------------------------------------------*/
		/*No Time Movement-move unitl reach limit sensor*/
		/*----------------------------------------------*/
		/*----------------------------*/
		case 499:
			/*----------------------------*/

			pMold->ActInfo.TopDeflashFw = 1;
			pMold->ActInfo.TopDeflashBw = 0;

			pMold->ValveOut.TopDeflashFw  = 1;
			pMold->ValveOut.TopDeflashBw  = 0;
			pMold->ValveOut.TopDeflashCls = 0;

			pMold->TopDeflash.p_set = pTopDeflashPara->P_Fw;/*Albert*/

			if(1 == pMold->TransDIn.TopDeflashFwLimit) /*2018.7.16 Albert*/
			{
				pMold->ValveOut.TopDeflashFw = 0;
				pMold->TopDeflash.Timer.IN   = 0;
				pMold->TopDeflash.LimitTimer.IN = 0;
				//	pMold->TimeDis.TopDeflashFwTime = 0;

				pMold->TopDeflash.p_set = 0;/*Albert*/
				if(1 == gMachineInfo.Auto)
				{
					pMold->TopDeflash.Step = 500;
				}
				else
				{
					pMold->TopDeflash.Step = 2900;
				}
			}

			pMold->TimeDis.TopDeflashFwAlarmTime = pMold->TopDeflash.LimitTimer.ET;

			if (1 == pMold->TopDeflash.LimitTimer.Q )
			{
				pMold->Alarm.TopDeflashNotAtFwPos=1;
				pMold->TopDeflash.Timer.IN   = 0;
				pMold->TopDeflash.LimitTimer.IN = 0;
				pMold->TopDeflash.Step = 40000;
			}

			break;

		/* ------------------------- handle forward ------------------------- */
		case 500:
			HandledeflashCount=0;
			if(pMold->Option.PunchHandle)
			{
				if(pMold->TimeSet.TopDeflashClsDelay != 0)
				{
					pMold->TopDeflash.Timer.IN = 1;
					pMold->TopDeflash.Timer.PT = pMold->TimeSet.TopDeflashClsDelay;
					pMold->TopDeflash.Step 	= 600;
				}
				else
				{
					pMold->TopDeflash.Step = 700;
				}
			}
			else
			{
				pMold->TopDeflash.Step = 900;
			}
			break;

		case 600:				/* handle delay ok */
			pMold->TimeDis.TopDeflashClsDelay = pMold->TopDeflash.Timer.ET;
			if (1 == pMold->TopDeflash.Timer.Q)
			{
				pMold->TopDeflash.Timer.IN        = 0;
				//	pMold->TimeDis.TopDeflashClsDelay = 0;
				pMold->TopDeflash.Step = 700;
			}
			break;

		case 700:
			if(pMold->TimeSet.TopDeflashClsTime != 0)
			{
				pMold->TopDeflash.Timer.IN = 1;
				pMold->TopDeflash.Timer.PT = pMold->TimeSet.TopDeflashClsTime;
				pMold->TopDeflash.Step = 800;
			}
			else
			{
				pMold->TopDeflash.Step = 900;
			}
			break;

		case 800:				/* TopDeflash handle time ok */

			pMold->ActInfo.TopDeflashFw    = 0;
			pMold->ActInfo.TopDeflashPuncher = 1;
			pMold->ActInfo.TopDeflashBw = 0;

			pMold->ValveOut.TopDeflashFw  = 0;
			pMold->ValveOut.TopDeflashCls = 1;

			pMold->TimeDis.TopDeflashClsTime = pMold->TopDeflash.Timer.ET;
			if (1 == pMold->TopDeflash.Timer.Q )
			{
				pMold->TopDeflash.Timer.IN = 0;
				//	pMold->TimeDis.TopDeflashClsTime = 0;

				//					if(1 == gMachineInfo.TimeLimit)
				//					{
				//						pMold->TopDeflash.Step = 900;
				//					}
				//					else
				//					{
				//						pMold->TopDeflash.Step = 2800;
				//					}
				pMold->TopDeflash.Step = 1100;

			}
			break;

		/* ------------------------- handle back ------------------------- */
		case 900:
			if(pMold->Option.PunchHandle)
			{
				if(pMold->TimeSet.TopDeflashOpnDelay != 0)
				{
					pMold->TopDeflash.Timer.IN = 1;
					pMold->TopDeflash.Timer.PT = pMold->TimeSet.TopDeflashOpnDelay;
					pMold->TopDeflash.Step 	= 1000;
				}
				else
				{
					pMold->TopDeflash.Step = 1100;
				}
			}
			else
			{
				pMold->TopDeflash.Step = 1100;
			}
			break;

		case 1000:
			pMold->TimeDis.TopDeflashOpnDelay = pMold->TopDeflash.Timer.ET;
			if (1 == pMold->TopDeflash.Timer.Q)
			{
				pMold->TopDeflash.Timer.IN        = 0;
				pMold->TimeDis.TopDeflashOpnDelay = 0;
				pMold->TopDeflash.Step = 1100;
			}
			break;

		case 1100:

			if (1==pMold->Option.PunchHandle)
			{
				pMold->TopDeflash.Timer.IN = 1;
				pMold->TopDeflash.Timer.PT = pMold->TimeSet.TopDeflashOpnAlarmTime;
				pMold->TopDeflash.Step = 1200;
			}
			else
			{
				//	pMold->TopDeflash.Step = 1210;
				pMold->TopDeflash.Step = 1300; //ipis0213
			}

			break;

		case 1200:

			pMold->ActInfo.TopDeflashFw    = 0;
			pMold->ActInfo.TopDeflashPuncher = 0;
			pMold->ActInfo.TopDeflashBw = 0;

			pMold->ValveOut.TopDeflashFw  = 0;
			pMold->ValveOut.TopDeflashBw  = 0;
			pMold->ValveOut.TopDeflashCls = 0;

			if (1 == pMold->TransDIn.TopDeflashOpnLimit)
			{
				pMold->TopDeflash.Timer.IN = 0;

				//				if(1==gMachineFix.Option.bHandledeflashRelpy )   /* Handledeflash 2 time*/
				//				{
				//					pMold->TopDeflash.Step = 1250;
				//				}
				//				else
				//				{
				//					pMold->TopDeflash.Step = 1300;
				//				}
				HandledeflashCount = HandledeflashCount+1;

				if (0==gUserPara.HandledeflashCount || (gUserPara.HandledeflashCount == HandledeflashCount))
				{
					HandledeflashCount=0;
					pMold->TopDeflash.Step = 1300;
				}
				else
				{
					pMold->TopDeflash.Step = 700;
				}

				//	pMold->TopDeflash.Step = 1300;

			}

			pMold->TimeDis.TopDeflashOpnAlarmTime = pMold->TopDeflash.Timer.ET;

			if(1 == pMold->TopDeflash.Timer.Q)
			{
				pMold->TopDeflash.Timer.IN = 0;
				pMold->Alarm.TopDeflashNotAtOpnPos = 1;
				pMold->TopDeflash.Step = 40000;           /*  TopDeflash backward alarm   */
			}
			break;

		case 1210: // for no use

			if (1 == pMold->TransDIn.TopDeflashOpnLimit)
			{
				pMold->TopDeflash.Timer.IN = 0;
				if(pMold->Option.TopDeflash)
				{
					pMold->TopDeflash.Step = 1300;		 // topdeflash bw
				}
				else
				{
					pMold->TopDeflash.Step = 3000;
				}

			}
			else
			{
				pMold->TopDeflash.Timer.IN = 0;
				pMold->Alarm.TopDeflashNotAtOpnPos = 1;
				pMold->TopDeflash.Step = 40000;           /*  TopDeflash backward alarm   */

			}

			break;

		case 1250:
			if(pMold->TimeSet.TopDeflashClsTime != 0)
			{
				pMold->TopDeflash.Timer.IN = 1;
				pMold->TopDeflash.Timer.PT = pMold->TimeSet.TopDeflashClsTime;
				pMold->TopDeflash.Step = 1260;
			}
			else
			{
				pMold->TopDeflash.Step = 1270;
			}
			break;

		case 1260:				/* TopDeflash handle time ok */

			pMold->ActInfo.TopDeflashFw    = 0;
			pMold->ActInfo.TopDeflashPuncher = 1;
			pMold->ActInfo.TopDeflashBw = 0;

			pMold->ValveOut.TopDeflashFw  = 1;
			pMold->ValveOut.TopDeflashCls = 1;

			pMold->TimeDis.TopDeflashClsTime = pMold->TopDeflash.Timer.ET;
			if (1 == pMold->TopDeflash.Timer.Q )
			{
				pMold->TopDeflash.Timer.IN = 0;
				//	pMold->TimeDis.TopDeflashClsTime = 0;

				pMold->TopDeflash.Step = 1270;

			}
			break;

		case 1270:
			pMold->TopDeflash.Timer.IN = 1;
			pMold->TopDeflash.Timer.PT = pMold->TimeSet.TopDeflashOpnAlarmTime;
			pMold->TopDeflash.Step = 1280;
			break;

		case 1280:
			pMold->ActInfo.TopDeflashFw    = 0;
			pMold->ActInfo.TopDeflashPuncher = 0;
			pMold->ActInfo.TopDeflashBw = 0;

			pMold->ValveOut.TopDeflashFw  = 0;
			pMold->ValveOut.TopDeflashBw  = 0;
			pMold->ValveOut.TopDeflashCls = 0;

			if (1 == pMold->TransDIn.TopDeflashOpnLimit)
			{
				pMold->TopDeflash.Timer.IN = 0;

				//	pMold->TopDeflash.Step = 2800;

				pMold->TopDeflash.Step = 1300;

			}

			pMold->TimeDis.TopDeflashOpnAlarmTime = pMold->TopDeflash.Timer.ET;

			if(1 == pMold->TopDeflash.Timer.Q)
			{
				pMold->TopDeflash.Timer.IN = 0;
				pMold->Alarm.TopDeflashNotAtOpnPos = 1;
				pMold->TopDeflash.Step = 40000;           /*  TopDeflash backward alarm   */
			}
			break;

		/* ------------------------- topdeflash backward ------------------------- */
		case 1300:
			if(pMold->Option.TopDeflash)
			{
				switch (pTopDeflashFix->eActuatorType)
				{
					/*-------------------------------------------------*/
					case ACTUATOR_HYD: /*1:Oil*/
						/*-------------------------------------------------*/
						if(pMold->TimeSet.TopDeflashBwDelay != 0)
						{
							pMold->TopDeflash.Timer.IN = 1;
							pMold->TopDeflash.Timer.PT = pMold->TimeSet.TopDeflashBwDelay;
							pMold->TopDeflash.Step = 1400;

							//gExSPC
							if(pMold == & LMold)
							{
								gExSPC[ExIndex].LMold.TopDeflashBwDelay = pMold->TimeSet.TopDeflashBwDelay/100.0;
							}
							else
							{
								gExSPC[ExIndex].RMold.TopDeflashBwDelay = pMold->TimeSet.TopDeflashBwDelay/100.0;
							}
						}
						else
						{
							pMold->TopDeflash.Step = 1500;
						}
						break;
					/*-------------------------------------------------*/
					case ACTUATOR_PNEU: /*2:Air*/
						/*-------------------------------------------------*/
						pMold->TopDeflash.Step = 1500;
						break;
				}
			}
			else
			{
				pMold->TopDeflash.Step = 1500;
			}
			break;

		case 1400:				/* TopDeflash backward delay ok */
			pMold->TimeDis.TopDeflashBwDelay = pMold->TopDeflash.Timer.ET;
			if (1 == pMold->TopDeflash.Timer.Q)
			{
				pMold->TopDeflash.Timer.IN       = 0;
				//	pMold->TimeDis.TopDeflashBwDelay = 0;
				pMold->TopDeflash.Step = 1500;
			}
			break;

		case 1500:
			if(pMold->Option.TopDeflash)
			{
				pMold->TopDeflash.LimitTimer.IN = 1; //ipis0213
				pMold->TopDeflash.LimitTimer.PT = pMold->TimeSet.TopDeflashBwAlarmTime;
				pMold->TopDeflash.Step = 1600;
			}
			else
			{
				pMold->TopDeflash.Step = 1700;   //for no use
			}
			break;

		case 1600:

			pMold->ActInfo.TopDeflashFw = 0;
			pMold->ActInfo.TopDeflashPuncher = 0;
			pMold->ActInfo.TopDeflashBw = 1;

			pMold->ValveOut.TopDeflashFw  = 0;
			pMold->ValveOut.TopDeflashBw  = 1;
			pMold->ValveOut.TopDeflashCls = 0;

			if(1 == gMachineInfo.MachineReset)  /* AutoReset  */
			{
				pMold->TopDeflash.p_set = pTopDeflashPara->P_BwReset;
				pMold->TopDeflash.v_set = pTopDeflashPara->V_BwReset;
			}
			else
			{
				pMold->TopDeflash.p_set = pTopDeflashPara->P_Bw;/*Albert*/
				pMold->TopDeflash.v_set = pTopDeflashPara->V_Bw;
			}

			if (1 == pMold->TransDIn.TopDeflashBwLimit)
			{
				pMold->ValveOut.TopDeflashFw  = 0;
				pMold->ValveOut.TopDeflashBw  = 0;
				pMold->ValveOut.TopDeflashCls = 0;

				pMold->CoolDeflash.Step =500;  //owen1021

				pMold->TopDeflash.p_set = 0;/*Albert*/
				pMold->TopDeflash.v_set = 0;

				pMold->TopDeflash.Timer.IN   = 0;
				pMold->TopDeflash.Step = 2900;

				//gExSPC
				if(pMold == & LMold)
				{
					gExSPC[ExIndex].LMold.tTopDeflashBw = pMold->TopDeflash.Timer.ET/100.0;
				}
				else
				{
					gExSPC[ExIndex].RMold.tTopDeflashBw = pMold->TopDeflash.Timer.ET/100.0;
				}
			}

			pMold->TimeDis.TopDeflashBwAlarmTime = pMold->TopDeflash.LimitTimer.ET;

			//			if(1 == pMold->TopDeflash.LimitTimer.Q)
			//			{
			//				pMold->ValveOut.TopDeflashFw  = 0;
			//				pMold->ValveOut.TopDeflashBw  = 0;
			//				pMold->ValveOut.TopDeflashCls = 0;
			//
			//				pMold->TopDeflash.Timer.IN   = 0;
			//				pMold->Alarm.TopDeflashNotAtBwPos = 1;
			//				pMold->TopDeflash.Step = 40000;           /*  TopDeflash backward alarm   */
			//			}
			break;

		case 1700: // for no use

			if (1 == pMold->TransDIn.TopDeflashBwLimit)
			{
				pMold->ValveOut.TopDeflashFw  = 0;
				pMold->ValveOut.TopDeflashBw  = 0;
				pMold->ValveOut.TopDeflashCls = 0;

				pMold->TopDeflash.p_set = 0;/*Albert*/

				pMold->TopDeflash.Timer.IN   = 0;
				pMold->TopDeflash.Step = 2900;
			}
			else
			{
				pMold->TopDeflash.Timer.IN   = 0;
				pMold->Alarm.TopDeflashNotAtBwPos = 1;
				pMold->TopDeflash.Step = 40000;           /*  TopDeflash backward alarm   */

			}
			pMold->TimeDis.TopDeflashBwAlarmTime = pMold->TopDeflash.LimitTimer.ET;

			//			if(1 == pMold->TopDeflash.Timer.Q)
			//			{
			//				pMold->ValveOut.TopDeflashFw  = 0;
			//				pMold->ValveOut.TopDeflashBw  = 0;
			//				pMold->ValveOut.TopDeflashCls = 0;
			//
			//				pMold->TopDeflash.Timer.IN   = 0;
			//				pMold->Alarm.TopDeflashNotAtBwPos = 1;
			//				pMold->TopDeflash.Step = 40000;           /*  TopDeflash backward alarm   */
			//			}

			break;

		/*----------for handle Top deflash force backward------------------------------*/
		case 1950: //for auto force backward

			pMold->TopDeflash.Timer.IN = 0;
			pMold->TopDeflash.LimitTimer.IN = 0;
			pMold->TopDeflash.Step = 2000;
			break;

		case 2000:
			// Top deflash Open
			if (1 == pMold->Option.PunchHandle)
			{
				pMold->TopDeflash.LimitTimer.IN = 1;
				pMold->TopDeflash.LimitTimer.PT = pMold->TimeSet.TopDeflashOpnAlarmTime;
				pMold->TopDeflash.Step = 2050;
			}
			else
			{
				pMold->TopDeflash.Step = 2100; //ipis0213
			}

			break;

		case 2050:

			pMold->ActInfo.TopDeflashFw    = 0;
			pMold->ActInfo.TopDeflashPuncher = 0;
			pMold->ActInfo.TopDeflashBw = 0;

			pMold->ValveOut.TopDeflashFw  = 0;
			pMold->ValveOut.TopDeflashBw  = 0;
			pMold->ValveOut.TopDeflashCls = 0;

			if (1 == pMold->TransDIn.TopDeflashOpnLimit)
			{
				pMold->TopDeflash.Timer.IN = 0;

				HandledeflashCount=0;
				pMold->TopDeflash.Step = 2100;

			}

			pMold->TimeDis.TopDeflashOpnAlarmTime = pMold->TopDeflash.LimitTimer.ET;

			if(1 == pMold->TopDeflash.LimitTimer.Q)
			{
				pMold->TopDeflash.LimitTimer.IN = 0;
				pMold->Alarm.TopDeflashNotAtOpnPos = 1;
				pMold->TopDeflash.Step = 40000;           /*  TopDeflash backward alarm   */
			}

			break;

		case 2100:
			// Top deflash backward

			if(pMold->Option.TopDeflash)
			{
				pMold->TopDeflash.LimitTimer.IN = 1;
				pMold->TopDeflash.LimitTimer.PT = pMold->TimeSet.TopDeflashBwAlarmTime;
				pMold->TopDeflash.Step = 2150;
			}
			else
			{
				pMold->TopDeflash.Step = 2900;   //for no use
			}

			break;

		case 2150:

			pMold->ActInfo.TopDeflashFw    = 0;
			pMold->ActInfo.TopDeflashPuncher = 0;
			pMold->ActInfo.TopDeflashBw = 1;

			pMold->ValveOut.TopDeflashFw  = 0;
			pMold->ValveOut.TopDeflashBw  = 1;
			pMold->ValveOut.TopDeflashCls = 0;

			pMold->TopDeflash.p_set = pTopDeflashPara->P_Bw;/*Albert*/
			pMold->TopDeflash.v_set = pTopDeflashPara->V_Bw;

			if (1 == pMold->TransDIn.TopDeflashBwLimit)
			{
				pMold->ValveOut.TopDeflashFw  = 0;
				pMold->ValveOut.TopDeflashBw  = 0;
				pMold->ValveOut.TopDeflashCls = 0;

				pMold->TopDeflash.p_set = 0;/*Albert*/
				pMold->TopDeflash.v_set = 0;

				pMold->TopDeflash.LimitTimer.IN   = 0;
				pMold->TopDeflash.Step = 2900;
			}

			pMold->TimeDis.TopDeflashBwAlarmTime = pMold->TopDeflash.LimitTimer.ET;

			if(1 == pMold->TopDeflash.Timer.Q)
			{
				pMold->ValveOut.TopDeflashFw  = 0;
				pMold->ValveOut.TopDeflashBw  = 0;
				pMold->ValveOut.TopDeflashCls = 0;

				pMold->TopDeflash.LimitTimer.IN   = 0;
				pMold->Alarm.TopDeflashNotAtBwPos = 1;
				pMold->TopDeflash.Step = 40000;           /*  TopDeflash backward alarm   */
			}

			break;

		/*----------------------------------------------------------------------------*/

		/* ------------------------- deflash off ------------------------- */

		case 2800:
			pMold->ValveOut.TopDeflashFw  = 0;
			pMold->ValveOut.TopDeflashBw  = 0;
			pMold->ValveOut.TopDeflashCls = 0;

			pMold->ActInfo.TopDeflashFw    = 0;
			pMold->ActInfo.TopDeflashPuncher = 0;
			pMold->ActInfo.TopDeflashBw = 0;

			pMold->TopDeflash.Timer.IN = 0;
			pMold->TopDeflash.Step = 3000;
			break;

		case 2900:
			if(1 == gMachineInfo.Auto)
			{
				//				if(pMold == &RMold)
				//				{
				//					RMold.Option.TopDeflash  = gMacOption.RTopDeflash;
				//					RMold.Option.PunchHandle = gMacOption.RPunchHandle;
				//				}
				//
				//				if(pMold == &LMold)
				//				{
				//					LMold.Option.TopDeflash  = gMacOption.LTopDeflash;
				//					LMold.Option.PunchHandle = gMacOption.LPunchHandle;
				//				}

				pMold->ValveOut.TopDeflashFw  = 0;
				pMold->ValveOut.TopDeflashBw  = 0;
				pMold->ValveOut.TopDeflashCls = 0;

				pMold->ActInfo.TopDeflashFw    = 0;
				pMold->ActInfo.TopDeflashPuncher = 0;
				pMold->ActInfo.TopDeflashBw = 0;

				/*Albert*/
				//				pMold->BlowDeflash.Step = 500;		/*  吹冷飞边结束  */
				//				pMold->CoolDeflash.Step = 500;		/*  cool deflash end  */ //ipis0731
				pMold->ChuteDeflashBlow.Step = 100;	/*  吹掉廢胚   */

			}
			else
			{
				pMold->ValveOut.TopDeflashFw  = 0;
				pMold->ValveOut.TopDeflashBw  = 0;
				pMold->ValveOut.TopDeflashCls = 0;

				pMold->ActInfo.TopDeflashFw    = 0;
				pMold->ActInfo.TopDeflashPuncher = 0;
				pMold->ActInfo.TopDeflashBw = 0;

			}

			pMold->TopDeflash.Timer.IN = 0;
			pMold->TopDeflash.LimitTimer.IN = 0;

			pMold->TopDeflash.p_set = 0;
			pMold->TopDeflash.v_set = 0;

			pMold->TopDeflash.Step = 3000;

			break;

		case 3000:
			break;

		case 5000:

			//			pMold->ActInfo.TopDeflashFw    = 1;
			//			pMold->ActInfo.TopDeflashPuncher = 0;
			//			pMold->ActInfo.TopDeflashBw = 0;
			//
			//			pMold->ValveOut.TopDeflashFw  = 1;
			//			pMold->ValveOut.TopDeflashBw  = 0;
			//			pMold->ValveOut.TopDeflashCls = 0;
			//			pMold->ValveOut.TopDeflashCool = 0;/*Albert*/
			//
			//			pMold->TopDeflash.p_set = pTopDeflashPara->P_CalibFw;/*Albert*/

			if(0 == pMold->TransDIn.TopDeflashFwLimit)
			{
				pMold->ActInfo.TopDeflashFw    = 1;
				pMold->ActInfo.TopDeflashPuncher = 0;
				pMold->ActInfo.TopDeflashBw = 0;

				pMold->ValveOut.TopDeflashFw  = 1;
				pMold->ValveOut.TopDeflashBw  = 0;
				pMold->ValveOut.TopDeflashCls = 0;
				pMold->ValveOut.TopDeflashCool = 0;/*Albert*/

				//	pMold->TopDeflash.p_set = pTopDeflashPara->P_CalibFw;/*Albert*/
				pMold->TopDeflash.p_set = pTopDeflashFix->pCalibMax;
				pMold->TopDeflash.v_set = pTopDeflashFix->vCalibMax;
			}
			else
			{
				pMold->ActInfo.TopDeflashFw    = 0;
				pMold->ActInfo.TopDeflashPuncher = 0;
				pMold->ActInfo.TopDeflashBw = 0;

				pMold->ValveOut.TopDeflashFw  = 0;
				pMold->ValveOut.TopDeflashBw  = 0;
				pMold->ValveOut.TopDeflashCls = 0;

				pMold->TopDeflash.p_set = 0;
				pMold->TopDeflash.v_set = 0;

				pMold->TopDeflash.Step = 20000;
			}

			break;

		case 8000:

			pMold->ActInfo.TopDeflashFw    = 0;
			pMold->ActInfo.TopDeflashPuncher = 0;
			pMold->ActInfo.TopDeflashBw = 0;

			pMold->ValveOut.TopDeflashFw  = 0;
			pMold->ValveOut.TopDeflashBw  = 1;
			pMold->ValveOut.TopDeflashCls = 0;
			break;

		case 15000:
			//
			//			pMold->ActInfo.TopDeflashBw    = 1;
			//			pMold->ActInfo.TopDeflashPuncher = 0;
			//			pMold->ActInfo.TopDeflashFw = 0;
			//
			//			pMold->ValveOut.TopDeflashFw  = 0;
			//			pMold->ValveOut.TopDeflashBw  = 1;
			//			pMold->ValveOut.TopDeflashCls = 0;
			//			pMold->ValveOut.TopDeflashCool = 0;/*Albert*/
			//
			//			//pMold->TopDeflash.p_set = pTopDeflashPara->P_Bw;/*Albert*/
			//			pMold->TopDeflash.p_set = pTopDeflashPara->P_CalibBw;/*Albert*/
			//

			if(0 == pMold->TransDIn.TopDeflashBwLimit)
			{
				pMold->ActInfo.TopDeflashBw    = 1;
				pMold->ActInfo.TopDeflashPuncher = 0;
				pMold->ActInfo.TopDeflashFw = 0;

				pMold->ValveOut.TopDeflashFw  = 0;
				pMold->ValveOut.TopDeflashBw  = 1;
				pMold->ValveOut.TopDeflashCls = 0;
				pMold->ValveOut.TopDeflashCool = 0;/*Albert*/

				//pMold->TopDeflash.p_set = pTopDeflashPara->P_Bw;/*Albert*/
				//	pMold->TopDeflash.p_set = pTopDeflashPara->P_CalibBw;/*Albert*/
				pMold->TopDeflash.p_set = pTopDeflashFix->pCalibZero;/*ipis20190131*/
				pMold->TopDeflash.v_set = pTopDeflashFix->vCalibZero;/*ipis20190131*/

			}
			else
			{

				pMold->ActInfo.TopDeflashBw    = 0;
				pMold->ActInfo.TopDeflashPuncher = 0;
				pMold->ActInfo.TopDeflashFw = 0;

				pMold->ValveOut.TopDeflashFw  = 0;
				pMold->ValveOut.TopDeflashBw  = 0;
				pMold->ValveOut.TopDeflashCls = 0;
				pMold->ValveOut.TopDeflashCool = 0;/*Albert*/

				pMold->TopDeflash.p_set = 0;/*Albert*/
				pMold->TopDeflash.v_set = 0;

				pMold->TopDeflash.Step = 20000;
			}

			break;

		/*--------------- Manual action stop -----------------*/
		case 20000:
			switch (pTopDeflashFix->eActuatorType)
			{
				/*-------------------------------------------------*/
				case ACTUATOR_HYD: /*1:Oil*/
					/*-------------------------------------------------*/

					pMold->ValveOut.TopDeflashFw  = 0;
					pMold->ValveOut.TopDeflashBw  = 0;
					pMold->ValveOut.TopDeflashCool = 0;/*Albert*/

					pMold->ActInfo.TopDeflashFw    = 0;
					pMold->ActInfo.TopDeflashPuncher = 0;
					pMold->ActInfo.TopDeflashBw = 0;

					pMold->TopDeflash.p_set = 0;
					pMold->TopDeflash.v_set = 0;
					break;
				/*-------------------------------------------------*/
				case ACTUATOR_PNEU: /*2:Air*/
					/*-------------------------------------------------*/

					break;
			}

			pMold->TopDeflash.Timer.IN   = 0;
			pMold->TopDeflash.LimitTimer.IN = 0;

			pMold->TopDeflash.Step 	 = 0;
			break;

		/*--------------- Instance stop -----------------*/
		case 30000:
			switch (pTopDeflashFix->eActuatorType)
			{
				/*-------------------------------------------------*/
				case ACTUATOR_HYD: /*1:Oil*/
					/*-------------------------------------------------*/

					pMold->ValveOut.TopDeflashFw  = 0;
					pMold->ValveOut.TopDeflashBw  = 0;
					pMold->ValveOut.TopDeflashCool = 0;/*Albert*/

					pMold->ActInfo.TopDeflashFw    = 0;
					pMold->ActInfo.TopDeflashPuncher = 0;
					pMold->ActInfo.TopDeflashBw = 0;

					pMold->TopDeflash.p_set = 0;
					pMold->TopDeflash.v_set = 0;
					break;
				/*-------------------------------------------------*/
				case ACTUATOR_PNEU: /*2:Air*/
					/*-------------------------------------------------*/

					break;
			}

			pMold->TopDeflash.Timer.IN   = 0;
			pMold->TopDeflash.LimitTimer.IN = 0;

			pMold->TopDeflash.Step     = 0;
			break;

		/*--------------- Error  stop -----------------*/
		case 40000:
			switch (pTopDeflashFix->eActuatorType)
			{
				/*-------------------------------------------------*/
				case ACTUATOR_HYD: /*1:Oil*/
					/*-------------------------------------------------*/

					pMold->ValveOut.TopDeflashFw  = 0;
					pMold->ValveOut.TopDeflashBw  = 0;
					pMold->ValveOut.TopDeflashCool = 0;/*Albert*/

					pMold->ActInfo.TopDeflashFw    = 0;
					pMold->ActInfo.TopDeflashPuncher = 0;
					pMold->ActInfo.TopDeflashBw = 0;

					pMold->TopDeflash.p_set = 0;
					pMold->TopDeflash.v_set = 0;
					break;
				/*-------------------------------------------------*/
				case ACTUATOR_PNEU: /*2:Air*/
					/*-------------------------------------------------*/

					break;
			}

			pMold->TopDeflash.Timer.IN   = 0;
			pMold->TopDeflash.LimitTimer.IN = 0;

			break;

		case 41000:
			switch (pTopDeflashFix->eActuatorType)
			{
				/*-------------------------------------------------*/
				case ACTUATOR_HYD: /*1:Oil*/
					/*-------------------------------------------------*/

					pMold->ValveOut.TopDeflashFw  = 0;
					pMold->ValveOut.TopDeflashBw  = 0;
					pMold->ValveOut.TopDeflashCool = 0;/*Albert*/

					pMold->ActInfo.TopDeflashFw    = 0;
					pMold->ActInfo.TopDeflashPuncher = 0;
					pMold->ActInfo.TopDeflashBw = 0;

					pMold->TopDeflash.p_set = 0;
					pMold->TopDeflash.v_set = 0;
					break;
				/*-------------------------------------------------*/
				case ACTUATOR_PNEU: /*2:Air*/
					/*-------------------------------------------------*/

					break;
			}

			pMold->TopDeflash.Timer.IN   = 0;
			pMold->TopDeflash.LimitTimer.IN = 0;

			break;
	}/* end of switch */

	/* ----------------- TopDeflash Fw / Bw timeout --------------------  */
	if(1 == pMold->TopDeflash.LimitTimer.Q && 1 == gMachineInfo.TimeLimit)
	{
		if(pMold->TopDeflash.Step < 500 && pMold->TopDeflash.Step > 300)		/* TopDeflash Fw  */
		{
			pMold->Alarm.TopDeflashNotAtFwPos = 1;
			pMold->CoolDeflash.Step =500; //ipis0731
		}

		if(pMold->TopDeflash.Step < 1700 && pMold->TopDeflash.Step > 1400)	/* TopDeflash Bw  */
		{
			pMold->Alarm.TopDeflashNotAtBwPos = 1;
		}

		pMold->TopDeflash.Timer.IN   = 0;
		pMold->TopDeflash.LimitTimer.IN = 0;
		pMold->TopDeflash.Step = 40000;

	}

	/* ----------------- TopDeflash action limit --------------------  */
	if((pMold->TopDeflash.Step > 100 && pMold->TopDeflash.Step < 500) /*|| (5000 == pMold->TopDeflash.Step) */)
	{
		if(0 == pMold->Clamp.ClsPos)
		{
			pMold->Alarm.ClampNotAtClsDI  = !pMold->Clamp.ClsPos;
			pMold->TopDeflash.Step = 40000;
		}

		if(0 == pMold->Carriage.BwPos)
		{
			pMold->Alarm.CarriageNotAtBwDI = !pMold->Carriage.BwPos;
			pMold->TopDeflash.Step = 40000;
		}

		if(0 == pMold->TransDIn.TopDeflashOpnLimit)
		{
			pMold->Alarm.TopDeflashNotAtOpnPos = !pMold->TransDIn.TopDeflashOpnLimit;
			pMold->TopDeflash.Step = 40000;
		}

		/* robot up or forward */
		//		if(0 == pMold->TransDIn.RobotUpLimit && 0 == pMold->TransDIn.RobotBwLimit)
		//		{
		//			pMold->Alarm.RobotNotAtUpPos = ! pMold->TransDIn.RobotUpLimit;
		//			pMold->Alarm.RobotNotAtBwPos = ! pMold->TransDIn.RobotBwLimit;
		//			pMold->TopDeflash.Step = 40000;
		//		}
		/*Chaoi*/
		if(1 == gMachineFix.Option.bRobotFwAfterTopdeflash)
		{
			if(0 == pMold->Robot.Transfer.BwPos)
			{
				pMold->Alarm.RobotNotAtBwPos = ! pMold->Robot.Transfer.BwPos;
				pMold->TopDeflash.Step = 40000;
			}
		}

		if (0 == pMold->TransDIn.TopDeflashOpnLimit )
		{
			pMold->Alarm.TopDeflashNotAtOpnPos = !pMold->TransDIn.TopDeflashOpnLimit;
			pMold->TopDeflash.Step = 40000;
		}
		/*----------------------------------------------------------*/

	}/* if(pMold->TopDeflash.Step > 100 && pMold->TopDeflash.Step < 900) */

	if((pMold->TopDeflash.Step > 1300 && pMold->TopDeflash.Step < 1700))
	{

		if (0 == pMold->TransDIn.TopDeflashOpnLimit )
		{
			pMold->Alarm.TopDeflashNotAtOpnPos = !pMold->TransDIn.TopDeflashOpnLimit;
			pMold->TopDeflash.Step = 40000;
		}

	}

}/*end of function */
```

#### tdeflash.var
```iecst
VAR
	HandledeflashCount : USINT;
END_VAR
```

### Program Logical/process/blowdef (ANSIC, version 1.00.0) - cooling deflash in pin

#### blowdeflash.c
```c
/********************************************************************
 * COPYRIGHT --  B&R China
 ********************************************************************
 * Program: blowdeflash
 * File: blowdeflash.c
 * Author: lijianjun
 * Created: March 06, 2013
 ********************************************************************
 * Implementation of program blowdeflash --- blowing air to  deflasher control
 ********************************************************************/

#include <bur/plctypes.h>

#ifdef _DEFAULT_INCLUDES
	#include <AsDefault.h>
#endif

/**************************************************************************************
                            Function Declarations
**************************************************************************************/

void BlowDeflash( Mold_typ * pMold);

/**************************************************************************************
     	        		I N I T U P  O F   T H E   T A S K
**************************************************************************************/
_INIT void init ( void )
 {
 	LMold.BlowDeflash.Step = 0;
 	RMold.BlowDeflash.Step = 0;
 } /* end of _INIT */

 /*************************************************************************************
        				C Y C L I C   P A R T   O F   T H E   T A S K
**************************************************************************************/

 _CYCLIC void cyclic ( void )
 {
	BlowDeflash(&LMold);
	BlowDeflash(&RMold);

	gMachineOut.LMold.BlowDeflash = LMold.BlowDeflash.Out;
	gMachineOut.RMold.BlowDeflash = RMold.BlowDeflash.Out;

 } /* end of _CYCLIC */

void BlowDeflash( Mold_typ * pMold)
{
    /* ------ step machine control ------ */
	 switch (pMold->BlowDeflash.Step)
    {
   		/*------------------ stop all the output ------------------*/
         case 0:
         	pMold->BlowDeflash.Out  	= 0;
         	pMold->ActInfo.BlowDeflash  = 0;
         	pMold->BlowDeflash.Timer.IN	= 0;
         	break;

   		/*------------------ BlowDeflash close -------------------- */
   		case 100: /* BlowDeflash delay*/
				if(pMold->TimeSet.BlowDeflashDelay != 0)
    			{
    				pMold->BlowDeflash.Timer.IN = 1;
			   	 	pMold->BlowDeflash.Timer.PT = pMold->TimeSet.BlowDeflashDelay;
    				pMold->BlowDeflash.Step = 200;
    			}
    			else
    			{
    				pMold->BlowDeflash.Step = 300;
    			}
          	break;
         case 200: /* delay ok */
         	pMold->TimeDis.BlowDeflashDelay = pMold->BlowDeflash.Timer.ET;
         	if (1 == pMold->BlowDeflash.Timer.Q)
         	{
         		pMold->BlowDeflash.Timer.IN     = 0;
         	//	pMold->TimeDis.BlowDeflashDelay = 0;
         		pMold->BlowDeflash.Step = 300;
         	}
         	break;
         case 300:
         	if(pMold->TimeSet.BlowDeflashTime != 0)
         	{
         		pMold->BlowDeflash.Timer.IN = 1;
		         pMold->BlowDeflash.Timer.PT = pMold->TimeSet.BlowDeflashTime;
		         pMold->BlowDeflash.Step = 400;
         	}
         	else
         	{
         		pMold->BlowDeflash.Step = 500;
         	}
         	break;
         case 400:
         	pMold->ActInfo.BlowDeflash = 1;
         	pMold->BlowDeflash.Out     = 1;

         	pMold->TimeDis.BlowDeflashTime = pMold->BlowDeflash.Timer.ET;
         	if (1 == pMold->BlowDeflash.Timer.Q)
         	{
         		pMold->BlowDeflash.Out      = 0;
         		pMold->BlowDeflash.Timer.IN = 0;
         	//	pMold->TimeDis.BlowDeflashTime = 0;
         		pMold->BlowDeflash.Step = 500;
         	}
         	break;
         case 500:
         	pMold->BlowDeflash.Timer.IN = 0;
         	pMold->BlowDeflash.Out     = 0;
         	pMold->ActInfo.BlowDeflash = 0;
         	pMold->BlowDeflash.Step = 3000;
         	break;
         case 3000:
         	break;

         case 20000:
         	pMold->BlowDeflash.Out      = 0;
				pMold->BlowDeflash.Timer.IN = 0;

				pMold->ActInfo.BlowDeflash = 0;
				pMold->BlowDeflash.Step    = 0;
	         break;

			case 30000:
				pMold->BlowDeflash.Out      = 0;
				pMold->BlowDeflash.Timer.IN = 0;

				pMold->ActInfo.BlowDeflash  = 0;
				pMold->BlowDeflash.Step     = 0;
				break;
	 }/* end of switch */
}/*end of function */
```

### Program Logical/process/cooldef (ANSIC, version 1.00.0) - cooling deflash in deflash

#### cooldef.c - Implementation code
```c
/********************************************************************
 * COPYRIGHT -- B&R China
 ********************************************************************
 * Program: cooldef
 * File: cooldef.c
 * Author: lij
 * Created: December 08, 2014
 ********************************************************************
 * Implementation of program cooldef
 ********************************************************************/

#include <bur/plctypes.h>

#ifdef _DEFAULT_INCLUDES
	#include <AsDefault.h>
#endif

/**************************************************************************************
                            Function Declarations
**************************************************************************************/

void CoolDeflash( Mold_typ * pMold);

/**************************************************************************************
     	        		I N I T U P  O F   T H E   T A S K
**************************************************************************************/
void _INIT DeflashCINIT(void)
{
	/* TODO: Add code here */
   LMold.CoolDeflash.Step = 0;
   RMold.CoolDeflash.Step = 0;
}

/*************************************************************************************
        				C Y C L I C   P A R T   O F   T H E   T A S K
**************************************************************************************/
void _CYCLIC DeflashCCYCLIC(void)
{
	/* TODO: Add code here */

   CoolDeflash(&LMold);
   CoolDeflash(&RMold);

   gMachineOut.LMold.CoolDeflash = LMold.CoolDeflash.Out;
   gMachineOut.RMold.CoolDeflash = RMold.CoolDeflash.Out;

}
/*************************************************************************************
        				E X I T   P A R T   O F   T H E   T A S K
**************************************************************************************/
void _EXIT DeflashCEXIT(void)
{
	/* TODO: Add code here */
}

void CoolDeflash( Mold_typ * pMold)
{
   /* ------ step machine control ------ */
	switch ( pMold->CoolDeflash.Step )
	{
		/*------------------ stop all the output ------------------*/
		case 0:
			pMold->CoolDeflash.Out  	 = 0;
			pMold->ActInfo.CoolDeflash  = 0;
			pMold->CoolDeflash.Timer.IN = 0;
			break;

		/*------------------ CoolDeflash close -------------------- */
		case 100: /* CoolDeflash delay*/
			if(pMold->TimeSet.CoolDeflashDelay != 0)
			{
				pMold->CoolDeflash.Timer.IN = 1;
				pMold->CoolDeflash.Timer.PT = pMold->TimeSet.CoolDeflashDelay;
				pMold->CoolDeflash.Step = 200;
			}
			else
			{
				//     pMold->CoolDeflash.Step = 300;
				pMold->CoolDeflash.Step = 450;  //ipis0731
			}
			break;

		case 200: /* delay ok */
			pMold->TimeDis.CoolDeflashDelay = pMold->CoolDeflash.Timer.ET;
			if (1 == pMold->CoolDeflash.Timer.Q)
			{
				pMold->CoolDeflash.Timer.IN     = 0;
				//   pMold->TimeDis.CoolDeflashDelay = 0;
				pMold->CoolDeflash.Step = 450;  //ipis0731
				//   pMold->CoolDeflash.Step = 300;
			}
			break;

		case 300:
			pMold->CoolDeflash.Timer.IN = 1;
			pMold->CoolDeflash.Timer.PT = pMold->TimeSet.CoolDeflashTime;
			pMold->CoolDeflash.Step = 400;

		case 400:
			pMold->ActInfo.CoolDeflash = 1;
			pMold->CoolDeflash.Out     = 1;
			pMold->TimeDis.CoolDeflashTime = pMold->CoolDeflash.Timer.ET;
			if (1 == pMold->CoolDeflash.Timer.Q)
			{
				pMold->CoolDeflash.Timer.IN     = 0;
				pMold->TimeDis.CoolDeflashTime = 0;
				pMold->CoolDeflash.Step = 500;
			}
			break;

		case 450:
			pMold->ActInfo.CoolDeflash = 1;
			pMold->CoolDeflash.Out     = 1;

			break;

		case 500:
			pMold->CoolDeflash.Timer.IN = 0;
			pMold->CoolDeflash.Out     = 0;
			pMold->ActInfo.CoolDeflash = 0;
			pMold->CoolDeflash.Step = 3000;
			break;

		case 3000:
			break;

		case 20000:
			pMold->CoolDeflash.Out      = 0;
			pMold->CoolDeflash.Timer.IN = 0;

			pMold->ActInfo.CoolDeflash = 0;
			pMold->CoolDeflash.Step    = 0;
			break;

		case 30000:
			pMold->CoolDeflash.Out      = 0;
			pMold->CoolDeflash.Timer.IN = 0;

			pMold->ActInfo.CoolDeflash  = 0;
			pMold->CoolDeflash.Step     = 0;
			break;
	}/* end of switch */
}/*end of function */
```

### Program Logical/process/cutneck (ANSIC, version 1.00.0) - cut neck

#### cutneck.c
```c
/********************************************************************
 * COPYRIGHT --  B&R
 ********************************************************************
 * Program: cutneck
 * File: cutneck.c
 * Author: lijianjun
 * Created: March 06, 2013
 ********************************************************************
 * Implementation of program cutneck --- cut neck control
 ********************************************************************/

#include <bur/plctypes.h>

#ifdef _DEFAULT_INCLUDES
	#include <AsDefault.h>
#endif

/**************************************************************************************
                            Function Declarations
**************************************************************************************/

void CutNeck( Mold_typ * pMold);

/**************************************************************************************
     	        		I N I T U P  O F   T H E   T A S K
**************************************************************************************/
_INIT void init ( void )
 {
 	LMold.CutNeck.Step = 30000;
 	RMold.CutNeck.Step = 30000;
 } /* end of _INIT */

 /*************************************************************************************
        				C Y C L I C   P A R T   O F   T H E   T A S K
**************************************************************************************/

 _CYCLIC void cyclic ( void )
 {
	LMold.TransDIn.CutNeckOpnLimit = gMachineIn.LMold.CutNeckOpnLimit = 1;
	RMold.TransDIn.CutNeckOpnLimit = gMachineIn.RMold.CutNeckOpnLimit = 1;

	if(!LMold.TimeSet.CutNeckOpnAlarmTime)LMold.TimeSet.CutNeckOpnAlarmTime = 1000;  /* 10s  */
	if(!RMold.TimeSet.CutNeckOpnAlarmTime)RMold.TimeSet.CutNeckOpnAlarmTime = 1000;  /* 10s  */

	CutNeck(&LMold);
	CutNeck(&RMold);

	gMachineOut.LMold.CutNeckCls = LMold.ValveOut.CutNeckCls;
	gMachineOut.RMold.CutNeckCls = RMold.ValveOut.CutNeckCls;

	gMachineOut.LMold.CutNeck    = LMold.ValveOut.CutNeck;
	gMachineOut.RMold.CutNeck    = RMold.ValveOut.CutNeck;

 } /* end of _CYCLIC */

void CutNeck( Mold_typ * pMold)
{

	 switch ( pMold->CutNeck.Step )
    {
   		/*------------------ stop all the output ------------------*/
         case 0:
         	pMold->CutNeck.Out = 0;

         	pMold->ActInfo.CutNeck    = 0;
         	pMold->ActInfo.CutNeckCls = 0;

         	pMold->CutNeck.Timer.IN	= 0;
         	break;

   		/*------------------ CutNeck forward -------------------- */
   		case 100: 					/* CutNeck forward delay*/
   			if(pMold->Option.CutNeck)
   			{
   				if(pMold->TimeSet.CutNeckClsDelay != 0)
    			   {
       				pMold->CutNeck.Timer.IN = 1;
   			      pMold->CutNeck.Timer.PT = pMold->TimeSet.CutNeckClsDelay;
       				pMold->CutNeck.Step = 200;
       			}
       			else
       			{
       				pMold->CutNeck.Step = 300;
       			}
       		}
       		else
       		{
       			pMold->CutNeck.Step = 3000;
       		}
          	break;
         case 200: 					/* CutNeck forward delay ok */
         	pMold->TimeDis.CutNeckClsDelay = pMold->CutNeck.Timer.ET;
         	if (1 == pMold->CutNeck.Timer.Q)
         	{
         		pMold->CutNeck.Timer.IN     = 0;
         		pMold->TimeDis.CutNeckClsDelay = 0;
         		pMold->CutNeck.Step = 300;
         	}
         	break;
         case 300:
         	if(pMold->TimeSet.CutNeckClsTime != 0)
         	{
         		pMold->CutNeck.Timer.IN = 1;
		         pMold->CutNeck.Timer.PT = pMold->TimeSet.CutNeckClsTime;
		         pMold->CutNeck.Step = 400;
         	}
         	else
         	{
         		pMold->CutNeck.Step = 500;
         	}
         	break;
         case 400:					/* CutNeck forward time ok */
         	pMold->ActInfo.CutNeck    = 0;
         	pMold->ActInfo.CutNeckCls = 1;

         	pMold->ValveOut.CutNeckCls = 1;
         	pMold->ValveOut.CutNeck    = 0;

         	pMold->CutNeck.Out = 1;

         	pMold->TimeDis.CutNeckClsTime = pMold->CutNeck.Timer.ET;
         	if (1 == pMold->CutNeck.Timer.Q)
         	{
         		pMold->CutNeck.Timer.IN = 0;
         		pMold->TimeDis.CutNeckClsTime = 0;
         		pMold->CutNeck.Step = 500;
         	}
         	break;
   		case 500: /* CutNeck delay*/
   			if(pMold->TimeSet.CutNeckDelay != 0)
   			{
   				pMold->CutNeck.Timer.IN = 1;
		         pMold->CutNeck.Timer.PT = pMold->TimeSet.CutNeckDelay;
   				pMold->CutNeck.Step = 600;
   			}
   			else
   			{
   				pMold->CutNeck.Step = 700;
   			}
          	break;
         case 600: 					/* CutNeck close delay ok */
         	pMold->TimeDis.CutNeckDelay = pMold->CutNeck.Timer.ET;
         	if (1 == pMold->CutNeck.Timer.Q)
         	{
         		pMold->CutNeck.Timer.IN     = 0;
         		pMold->TimeDis.CutNeckDelay = 0;
         		pMold->CutNeck.Step = 700;
         	}
         	break;
         case 700:
         	if(pMold->TransDIn.RobotOpnLimit)			/*  机械手开位   */
         	{
             	if(pMold->TimeSet.CutNeckTime != 0)
             	{
             		pMold->CutNeck.Timer.IN = 1;
   			      pMold->CutNeck.Timer.PT = pMold->TimeSet.CutNeckTime;
   			      pMold->CutNeck.Step = 800;
             	}
             	else
             	{
             		pMold->CutNeck.Step = 900;
             	}
            }
         	break;
         case 800:
         	pMold->ActInfo.CutNeck    = 1;
         	pMold->ActInfo.CutNeckCls = 1;

         	pMold->ValveOut.CutNeckCls = 1;
         	pMold->ValveOut.CutNeck    = 1;

         	pMold->CutNeck.Out = 2;

         	pMold->TimeDis.CutNeckTime = pMold->CutNeck.Timer.ET;
         	if (1 == pMold->CutNeck.Timer.Q)
         	{
         		pMold->ValveOut.CutNeck    = 0;
		         pMold->CutNeck.Out = 0;

         		pMold->CutNeck.Timer.IN    = 0;
         		pMold->TimeDis.CutNeckTime = 0;
         		pMold->CutNeck.Step = 900;
         	}
         	break;
         case 900:
         	if(pMold->TimeSet.CutNeckOpnDelay != 0)
    		   {
   				pMold->CutNeck.Timer.IN = 1;
		         pMold->CutNeck.Timer.PT = pMold->TimeSet.CutNeckOpnDelay;
   				pMold->CutNeck.Step = 1000;
   			}
   			else
   			{
   				pMold->CutNeck.Step = 1100;
   			}
         	break;
         case 1000:
         	pMold->ActInfo.CutNeckCls = 0;
         	pMold->ActInfo.CutNeck    = 1;

         	pMold->ValveOut.CutNeckCls = 0;
         	pMold->ValveOut.CutNeck    = 1;

         	pMold->CutNeck.Out = 3;

         	pMold->TimeDis.CutNeckOpnDelay = pMold->CutNeck.Timer.ET;
         	if (1 == pMold->CutNeck.Timer.Q)
         	{
         		pMold->ValveOut.CutNeckCls = 0;
         		pMold->CutNeck.Timer.IN    = 0;
         		pMold->TimeDis.CutNeckOpnDelay = 0;
         		pMold->CutNeck.Step = 1100;
         	}
         	break;
         case 1100:
         	pMold->CutNeck.Timer.IN = 1;
	         pMold->CutNeck.Timer.PT = pMold->TimeSet.CutNeckOpnAlarmTime;
	         pMold->CutNeck.Step = 1200;
         	break;
         case 1200:
         	pMold->ActInfo.CutNeckCls = 0;
         	pMold->ActInfo.CutNeck    = 0;

	         pMold->CutNeck.Out = 0;

         	pMold->ValveOut.CutNeckCls = 0;
         	pMold->ValveOut.CutNeck    = 0;

         	if(pMold->TransDIn.CutNeckOpnLimit)
         	{
         		pMold->CutNeck.Timer.IN = 0;
         		pMold->CutNeck.Step     = 1300;
         	}
         	pMold->TimeDis.CutNeckOpnAlarmTime = pMold->CutNeck.Timer.ET;
         	if (1 == pMold->CutNeck.Timer.Q)
         	{
         		pMold->CutNeck.Timer.IN = 0;
         		pMold->Alarm.CutNeckFwNotAtOpnPos = 1;
         		pMold->CutNeck.Step = 40000;
         	}
         	break;
         case 1300:
         	pMold->ActInfo.CutNeckCls = 0;
         	pMold->ActInfo.CutNeck    = 0;

         	pMold->ValveOut.CutNeckCls = 0;
         	pMold->ValveOut.CutNeck    = 0;

	         pMold->CutNeck.Out = 0;

         	pMold->CutNeck.Timer.IN = 0;
         	pMold->ActInfo.CutNeck  = 0;
         	pMold->CutNeck.Step = 3000;
         	break;
         case 3000:
         	break;

         /*--------------- Manual action stop -----------------*/
         case 20000:
         	pMold->ValveOut.CutNeckCls = 0;
         	pMold->ValveOut.CutNeck    = 0;

         	pMold->CutNeck.Out      = 0;
	         pMold->CutNeck.Timer.IN = 0;

         	pMold->ActInfo.CutNeckCls = 0;
         	pMold->ActInfo.CutNeck    = 0;

	         pMold->CutNeck.Step    = 0;
	         break;

			/*--------------- Instance stop -----------------*/
			case 30000:
	         pMold->ValveOut.CutNeckCls = 0;
         	pMold->ValveOut.CutNeck    = 0;

	         pMold->CutNeck.Out      = 0;
         	pMold->CutNeck.Timer.IN = 0;

         	pMold->ActInfo.CutNeckCls = 0;
         	pMold->ActInfo.CutNeck    = 0;

	         pMold->CutNeck.Step     = 0;
	         break;

         /*--------------- Error  stop -----------------*/
         case 40000:
         	pMold->ValveOut.CutNeckCls = 0;
         	pMold->ValveOut.CutNeck    = 0;

	         pMold->CutNeck.Out      = 0;
	         pMold->CutNeck.Timer.IN = 0;

         	pMold->ActInfo.CutNeckCls = 0;
         	pMold->ActInfo.CutNeck    = 0;
	         break;
	 }/* end of switch */

	if(pMold->CutNeck.Step > 100 && pMold->CutNeck.Step < 1300)
	{
	 	if(!pMold->Option.CutNeck && 1 == gMachineInfo.Auto)
	 	{
			pMold->CutNeck.Step = 1300;
		}
	}
}/*end of function */
```

### Program Logical/process/inerpin (ANSIC, version 1.00.0) - inner pin

#### innerpin.c
```c
/********************************************************************
 * COPYRIGHT --  B&R
 ********************************************************************
 * Program: inerpin
 * File: inerpin.c
 * Author: lijianjun
 * Created: March 06, 2013
 ********************************************************************
 * Implementation of program inerpin ---inner pin  control
 ********************************************************************/

#include <bur/plctypes.h>

#ifdef _DEFAULT_INCLUDES
	#include <AsDefault.h>
#endif

/**************************************************************************************
                            Function Declarations
**************************************************************************************/

void InnerPin( Mold_typ * pMold);

/**************************************************************************************
     	        		I N I T U P  O F   T H E   T A S K
**************************************************************************************/
_INIT void init ( void )
 {
 	LMold.InnerPin.Step = 0;
 	RMold.InnerPin.Step = 0;
 } /* end of _INIT */

 /*************************************************************************************
        				C Y C L I C   P A R T   O F   T H E   T A S K
**************************************************************************************/

 _CYCLIC void cyclic ( void )
 {
 	if(!LMold.TimeSet.InnerPinBwAlarmTime)LMold.TimeSet.InnerPinBwAlarmTime = 1000;
 	if(!RMold.TimeSet.InnerPinBwAlarmTime)RMold.TimeSet.InnerPinBwAlarmTime = 1000;

 	LMold.TransDIn.InnerPinBwLimit = gMachineIn.LMold.InnerPinBwLimit;
	RMold.TransDIn.InnerPinBwLimit = gMachineIn.RMold.InnerPinBwLimit;

	InnerPin(&LMold);
	InnerPin(&RMold);

	switch(LMold.InnerPin.Out)
	{
		case 0:
			gMachineOut.LMold.InnerPinFw   = 0;
			gMachineOut.LMold.InnerPinBlow = 0;
			break;
		case 1:
			gMachineOut.LMold.InnerPinFw   = 1;
			gMachineOut.LMold.InnerPinBlow = 0;
			break;
		case 2:
			gMachineOut.LMold.InnerPinFw   = 1;
			gMachineOut.LMold.InnerPinBlow = 1;
			break;
	}/* switch(LMold.InnerPin.Out) */

	switch(RMold.InnerPin.Out)
	{
		case 0:
			gMachineOut.RMold.InnerPinFw   = 0;
			gMachineOut.RMold.InnerPinBlow = 0;
			break;
		case 1:
			gMachineOut.RMold.InnerPinFw   = 1;
			gMachineOut.RMold.InnerPinBlow = 0;
			break;
		case 2:
			gMachineOut.RMold.InnerPinFw   = 1;
			gMachineOut.RMold.InnerPinBlow = 1;
			break;
	}/* switch(LMold.InnerPin.Out) */

 } /* end of _CYCLIC */

void InnerPin( Mold_typ * pMold)
{
   /* ------ step machine control ----- */
	switch ( pMold->InnerPin.Step )
   {
   		/*------------------ stop all the output ------------------*/
         case 0:
         	pMold->InnerPin.Out  	 = 0;
         	pMold->ActInfo.InnerPin  = 0;
         	pMold->InnerPin.Timer.IN = 0;
         	break;

   		/*------------------ InnerPin close -------------------- */
   		case 100: /* InnerPin delay*/
   			if(pMold->Option.InnerPin)
   			{
   				if(pMold->TimeSet.InnerPinFwDelay != 0)
       			{
       				pMold->InnerPin.Timer.IN = 1;
   			      pMold->InnerPin.Timer.PT = pMold->TimeSet.InnerPinFwDelay;
       				pMold->InnerPin.Step = 200;
       			}
       			else
       			{
       				pMold->InnerPin.Step = 300;
       			}
       		}
       		else
       		{
       			pMold->InnerPin.Step = 3000;
       		}
          	break;
         case 200: /* delay ok */
         	pMold->TimeDis.InnerPinFwDelay = pMold->InnerPin.Timer.ET;
         	if (1 == pMold->InnerPin.Timer.Q)
         	{
         		pMold->InnerPin.Timer.IN     = 0;
         		pMold->TimeDis.InnerPinFwDelay = 0;
         		pMold->InnerPin.Step = 300;
         	}
         	break;
         case 300:
         	pMold->ActInfo.InnerPin = 1;
         	pMold->InnerPin.Out     = 1;
	         pMold->InnerPin.Step = 3000;
         	break;

         /*case 300:
         	if(pMold->TimeSet.InnerPinFwTime != 0)
         	{
         		pMold->InnerPin.Timer.IN = 1;
		         pMold->InnerPin.Timer.PT = pMold->TimeSet.InnerPinFwTime;
		         pMold->InnerPin.Step = 400;
         	}
         	else
         	{
         		pMold->InnerPin.Step = 500;
         	}
         	break;
         case 400:
         	pMold->ActInfo.InnerPin = 1;
         	pMold->InnerPin.Out     = 1;
         	pMold->TimeDis.InnerPinFwTime = pMold->InnerPin.Timer.ET;
         	if (1 == pMold->InnerPin.Timer.Q)
         	{
         		pMold->InnerPin.Timer.IN = 0;
         		pMold->TimeDis.InnerPinFwTime = 0;
         		pMold->InnerPin.Step = 500;
         	}
         	break;
         case 500:
         	if(pMold->TimeSet.InnerPinBlowDelay != 0)
    		   {
   				pMold->InnerPin.Timer.IN = 1;
		         pMold->InnerPin.Timer.PT = pMold->TimeSet.InnerPinBlowDelay;
   				pMold->InnerPin.Step = 600;
   			}
   			else
   			{
   				pMold->InnerPin.Step = 700;
   			}
         	break;
         case 600:
         	pMold->TimeDis.InnerPinBlowDelay = pMold->InnerPin.Timer.ET;
         	if (1 == pMold->InnerPin.Timer.Q)
         	{
         		pMold->InnerPin.Timer.IN     = 0;
         		pMold->TimeDis.InnerPinBlowDelay = 0;
         		pMold->InnerPin.Step = 300;
         	}
         	break;
         case 700:
         	if(pMold->TimeSet.InnerPinBlowTime != 0)
    		   {
   				pMold->InnerPin.Timer.IN = 1;
		         pMold->InnerPin.Timer.PT = pMold->TimeSet.InnerPinBlowTime;
   				pMold->InnerPin.Step = 800;
   			}
   			else
   			{
   				pMold->InnerPin.Step = 900;
   			}
         	break;
         case 800:
         	pMold->ActInfo.InnerPin = 1;
         	pMold->InnerPin.Out     = 2;
         	pMold->TimeDis.InnerPinBlowTime = pMold->InnerPin.Timer.ET;
         	if (1 == pMold->InnerPin.Timer.Q)
         	{
         		pMold->InnerPin.Out      = 0;
         		pMold->InnerPin.Timer.IN = 0;
         		pMold->TimeDis.InnerPinBlowTime = 0;
         		pMold->InnerPin.Step = 900;
         	}
         	break;
         case 900:
         	pMold->InnerPin.Timer.IN = 0;
         	pMold->InnerPin.Out     = 0;
         	pMold->ActInfo.InnerPin = 0;
         	pMold->InnerPin.Step = 3000;
         	break;*/
         case 3000:
         	break;

         case 10100: 	/* InnerPin backward delay*/
   			if(pMold->Option.InnerPin)
   			{
   				if(pMold->TimeSet.InnerPinBwDelay != 0)
       			{
       				pMold->InnerPin.Timer.IN = 1;
   			      pMold->InnerPin.Timer.PT = pMold->TimeSet.InnerPinBwDelay;
       				pMold->InnerPin.Step = 10200;
       			}
       			else
       			{
       				pMold->InnerPin.Step = 10300;
       			}
    		   }
    		   else
    		   {
    			   pMold->InnerPin.Step = 13000;
    		   }
          	break;
         case 10200: 	/* backward delay ok */
         	pMold->TimeDis.InnerPinBwDelay = pMold->InnerPin.Timer.ET;
         	if (1 == pMold->InnerPin.Timer.Q)
         	{
         		pMold->InnerPin.Timer.IN     = 0;
         		pMold->TimeDis.InnerPinBwDelay = 0;
         		pMold->InnerPin.Step = 10300;
         	}
         	break;
         case 10300:
         	pMold->InnerPin.Timer.IN = 1;
	         pMold->InnerPin.Timer.PT = pMold->TimeSet.InnerPinBwAlarmTime;
    		   pMold->InnerPin.Step = 10400;
         	break;
			case 10400:
				pMold->ActInfo.InnerPin = 0;
				pMold->InnerPin.Out     = 0;

				if(pMold->TransDIn.InnerPinBwLimit)
				{
					pMold->InnerPin.Timer.IN = 0;
					pMold->InnerPin.Step = 13000;
				}

				pMold->TimeDis.InnerPinBwAlarmTime = pMold->InnerPin.Timer.ET;

				if (1 == pMold->InnerPin.Timer.Q)
				{
					pMold->Alarm.InnerPinNotAtBwPos = 1;
					pMold->InnerPin.Step = 40000;
				}
				break;
			case 13000:
				break;

			/*  normal stop  */
         case 20000:
            pMold->InnerPin.Out      = 0;
				pMold->InnerPin.Timer.IN = 0;

				pMold->ActInfo.InnerPin = 0;
				pMold->InnerPin.Step    = 0;
				break;

			/*--------------- Instancy stop -----------------*/
			case 30000:
				pMold->InnerPin.Out      = 0;
				pMold->InnerPin.Timer.IN = 0;

				pMold->ActInfo.InnerPin  = 0;
				pMold->InnerPin.Step     = 0;
				break;

			/*--------------- Error stop -----------------*/
			case 40000:
				pMold->InnerPin.Out      = 0;
				pMold->InnerPin.Timer.IN = 0;

				pMold->ActInfo.InnerPin  = 0;
				break;
	 }/* end of switch */

	if(pMold->InnerPin.Step > 100 && pMold->InnerPin.Step < 900)
	{
	 	if(!pMold->Option.InnerPin && 1 == gMachineInfo.Auto)
	 	{
			pMold->InnerPin.Step  = 20000;
		}
	}

}/*end of function */
```

### Program Logical/process/pullbottom (ANSIC, version 1.00.0) - pull bottom
